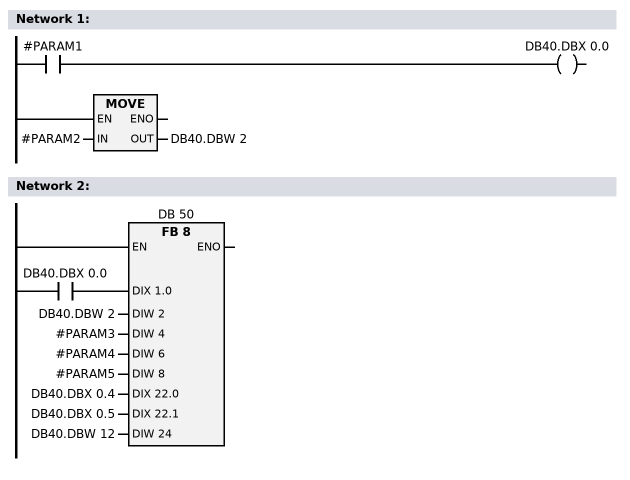
NETWORK
TITLE =
      A     #PARAM1;
      =     DB40.DBX 0.0;
      L     #PARAM2;
      T     DB40.DBW 2;
NETWORK
TITLE =
      A     DB40.DBX 0.0;
      =     L 0.0;
      BLD   103;
      CALL  FB 8 , DB 50 (
           DIX 1.0                  := L 0.0,
           DIW 2                    := DB40.DBW 2,
           DIW 4                    := #PARAM3,
           DIW 6                    := #PARAM4,
           DIW 8                    := #PARAM5,
           DIX 22.0                 := DB40.DBX 0.4,
           DIX 22.1                 := DB40.DBX 0.5,
           DIW 24                   := DB40.DBW 12);
      NOP   0;
NETWORK
TITLE =
      AN    DB40.DBX 0.4;
      JC    M001;
      L     DB40.DBW 16;
      +     1;
      T     DB40.DBW 16;
      NOP   0;
      NOP   0;
      NOP   0;
      BE;
M001: AN    DB40.DBX 0.5;
      BEC;
      L     DB40.DBW 18;
      +     1;
      T     DB40.DBW 18;
      L     DB40.DBW 12;
      T     DB40.DBW 14;
      NOP   0;
      NOP   0;
      NOP   0;
      BE;
NETWORK
TITLE =
END_FUNCTION

FUNCTION FC 31 : VOID
VERSION : 0.1
BEGIN
// (block stored without names or comments; labels and parameter names are numbered)
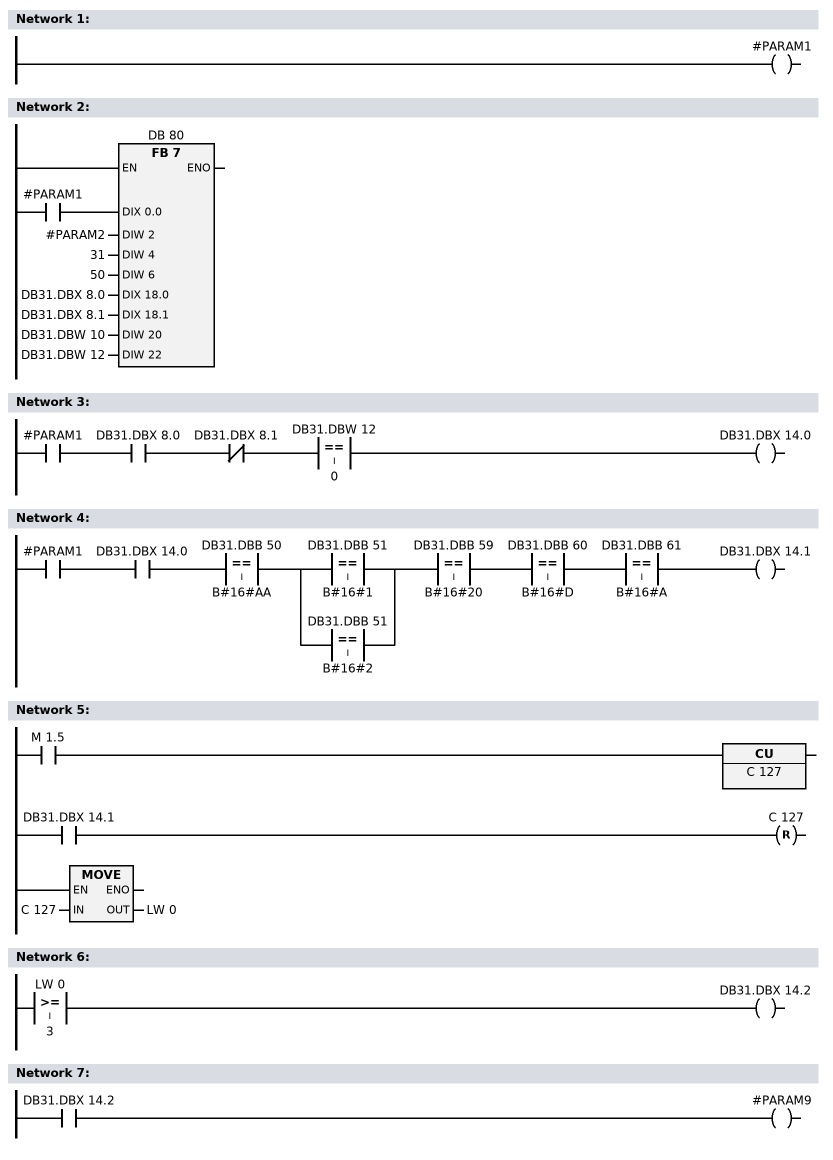
NETWORK
TITLE =
      SET;
      =     #PARAM1;
NETWORK
TITLE =
      A     #PARAM1;
      =     L 4.0;
      BLD   103;
      CALL  FB 7 , DB 80 (
           DIX 0.0                  := L 4.0,
           DIW 2                    := #PARAM2,
           DIW 4                    := 31,
           DIW 6                    := 50,
           DIX 18.0                 := DB31.DBX 8.0,
           DIX 18.1                 := DB31.DBX 8.1,
           DIW 20                   := DB31.DBW 10,
           DIW 22                   := DB31.DBW 12);
      NOP   0;
NETWORK
TITLE =
      A     #PARAM1;
      A     DB31.DBX 8.0;
      AN    DB31.DBX 8.1;
      A(;
      L     DB31.DBW 12;
      L     0;
      ==I;
      );
      =     DB31.DBX 14.0;
NETWORK
TITLE =
      A     #PARAM1;
      A     DB31.DBX 14.0;
      A(;
      L     DB31.DBB 50;
      L     B#16#AA;
      ==I;
      );
      A(;
      O(;
      L     DB31.DBB 51;
      L     B#16#1;
      ==I;
      );
      O(;
      L     DB31.DBB 51;
      L     B#16#2;
      ==I;
      );
      );
      A(;
      L     DB31.DBB 59;
      L     B#16#20;
      ==I;
      );
      A(;
      L     DB31.DBB 60;
      L     B#16#D;
      ==I;
      );
      A(;
      L     DB31.DBB 61;
      L     B#16#A;
      ==I;
      );
      =     DB31.DBX 14.1;
NETWORK
TITLE =
      A     M 1.5;
      CU    C 127;
      BLD   101;
      NOP   0;
      NOP   0;
      A     DB31.DBX 14.1;
      R     C 127;
      L     C 127;
      T     LW 0;
      NOP   0;
      NOP   0;
NETWORK
TITLE =
      L     LW 0;
      L     3;
      >=I;
      =     DB31.DBX 14.2;
NETWORK
TITLE =
      A     DB31.DBX 14.2;
      =     #PARAM9;
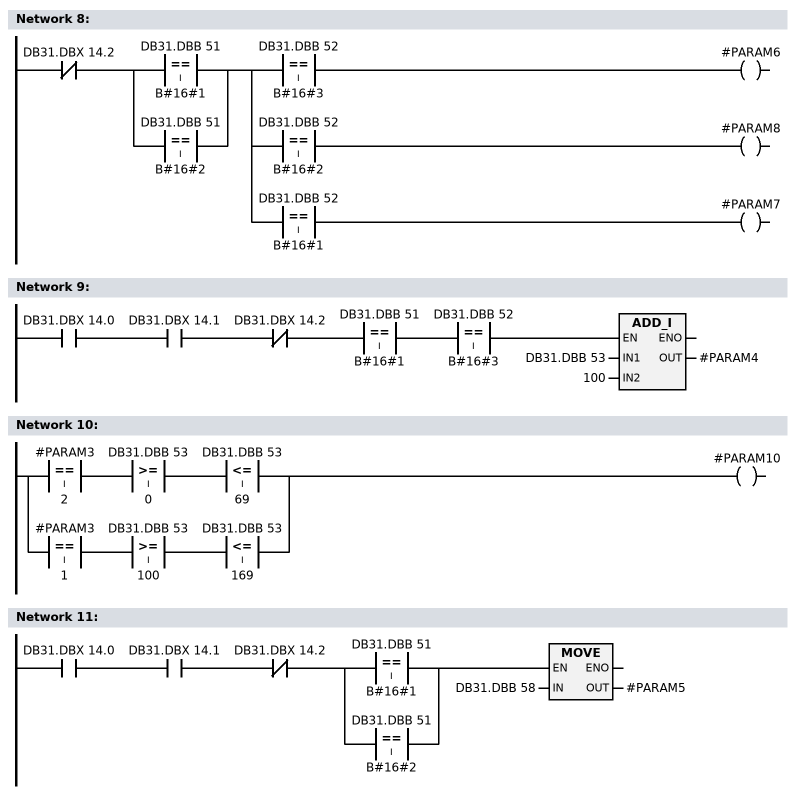
NETWORK
TITLE =
      AN    DB31.DBX 14.2;
      A(;
      O(;
      L     DB31.DBB 51;
      L     B#16#1;
      ==I;
      );
      O(;
      L     DB31.DBB 51;
      L     B#16#2;
      ==I;
      );
      );
      =     L 2.0;
      A     L 2.0;
      A(;
      L     DB31.DBB 52;
      L     B#16#3;
      ==I;
      );
      =     #PARAM6;
      A     L 2.0;
      A(;
      L     DB31.DBB 52;
      L     B#16#2;
      ==I;
      );
      =     #PARAM8;
      A     L 2.0;
      A(;
      L     DB31.DBB 52;
      L     B#16#1;
      ==I;
      );
      =     #PARAM7;
NETWORK
TITLE =
      A     DB31.DBX 14.0;
      A     DB31.DBX 14.1;
      AN    DB31.DBX 14.2;
      A(;
      L     DB31.DBB 51;
      L     B#16#1;
      ==I;
      );
      A(;
      L     DB31.DBB 52;
      L     B#16#3;
      ==I;
      );
      JNB   M001;
      L     DB31.DBB 53;
      L     100;
      +I;
      T     #PARAM4;
M001: NOP   0;
NETWORK
TITLE =
      A(;
      L     #PARAM3;
      L     2;
      ==I;
      );
      A(;
      L     DB31.DBB 53;
      L     0;
      >=I;
      );
      A(;
      L     DB31.DBB 53;
      L     69;
      <=I;
      );
      O;
      A(;
      L     #PARAM3;
      L     1;
      ==I;
      );
      A(;
      L     DB31.DBB 53;
      L     100;
      >=I;
      );
      A(;
      L     DB31.DBB 53;
      L     169;
      <=I;
      );
      =     #PARAM10;
NETWORK
TITLE =
      A     DB31.DBX 14.0;
      A     DB31.DBX 14.1;
      AN    DB31.DBX 14.2;
      A(;
      O(;
      L     DB31.DBB 51;
      L     B#16#1;
      ==I;
      );
      O(;
      L     DB31.DBB 51;
      L     B#16#2;
      ==I;
      );
      );
      JNB   M002;
      L     DB31.DBB 58;
      T     #PARAM5;
M002: NOP   0;
NETWORK
TITLE =
      A     DB31.DBX 8.0;
      JCN   M003;
      L     DB31.DBW 18;
      +     1;
      T     DB31.DBW 18;
      L     DB31.DBW 10;
      T     DB31.DBW 16;
      JU    M005;
M003: A     DB31.DBX 8.1;
      JCN   M004;
      L     DB31.DBW 20;
      +     1;
      T     DB31.DBW 20;
      L     0;
      L     DB31.DBW 12;
      ==I;
      JC    M005;
      T     DB31.DBW 22;
      JU    M005;
M004: L     0;
      L     DB31.DBW 12;
      ==I;
      JC    M005;
      T     DB31.DBW 22;
M005: CLR;
END_FUNCTION

FUNCTION FC 32 : VOID
VERSION : 0.1
BEGIN
// (block stored without names or comments; labels and parameter names are numbered)
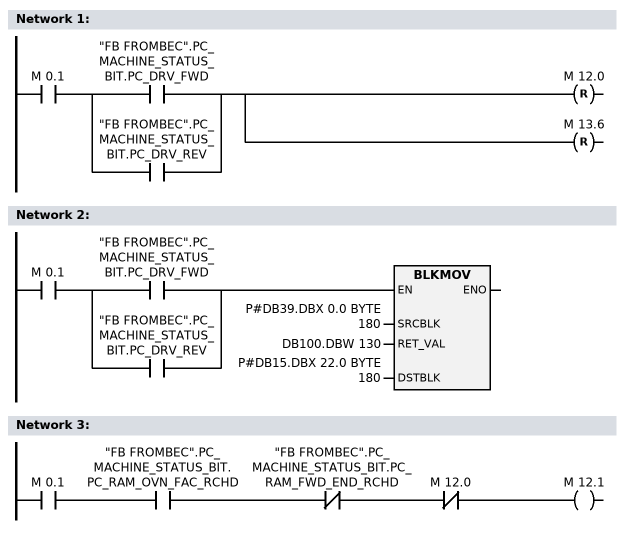
NETWORK
TITLE =
      A     M 0.1;
      A(;
      O     "FB FROMBEC".PC_MACHINE_STATUS_BIT.PC_DRV_FWD;
      O     "FB FROMBEC".PC_MACHINE_STATUS_BIT.PC_DRV_REV;
      );
      R     M 12.0;
      R     M 13.6;
NETWORK
TITLE =
      A     M 0.1;
      A(;
      O     "FB FROMBEC".PC_MACHINE_STATUS_BIT.PC_DRV_FWD;
      O     "FB FROMBEC".PC_MACHINE_STATUS_BIT.PC_DRV_REV;
      );
      JNB   M001;
      CALL  "BLKMOV" (
           SRCBLK                   := P#DB39.DBX 0.0 BYTE 180,
           RET_VAL                  := DB100.DBW 130,
           DSTBLK                   := P#DB15.DBX 22.0 BYTE 180);
M001: NOP   0;
NETWORK
TITLE =
      A     M 0.1;
      A     "FB FROMBEC".PC_MACHINE_STATUS_BIT.PC_RAM_OVN_FAC_RCHD;
      AN    "FB FROMBEC".PC_MACHINE_STATUS_BIT.PC_RAM_FWD_END_RCHD;
      AN    M 12.0;
      =     M 12.1;
NETWORK
TITLE =
      A(;
      A     M 0.1;
      A     M 12.1;
      A     M 1.3;
      FP    M 12.5;
      CU    C 120;
      BLD   101;
      NOP   0;
      NOP   0;
      A     M 12.0;
      R     C 120;
      L     C 120;
      T     MW 10;
      NOP   0;
      A     C 120;
      );
      A(;
      L     MW 10;
      L     91;
      ==I;
      );
      S     M 12.0;
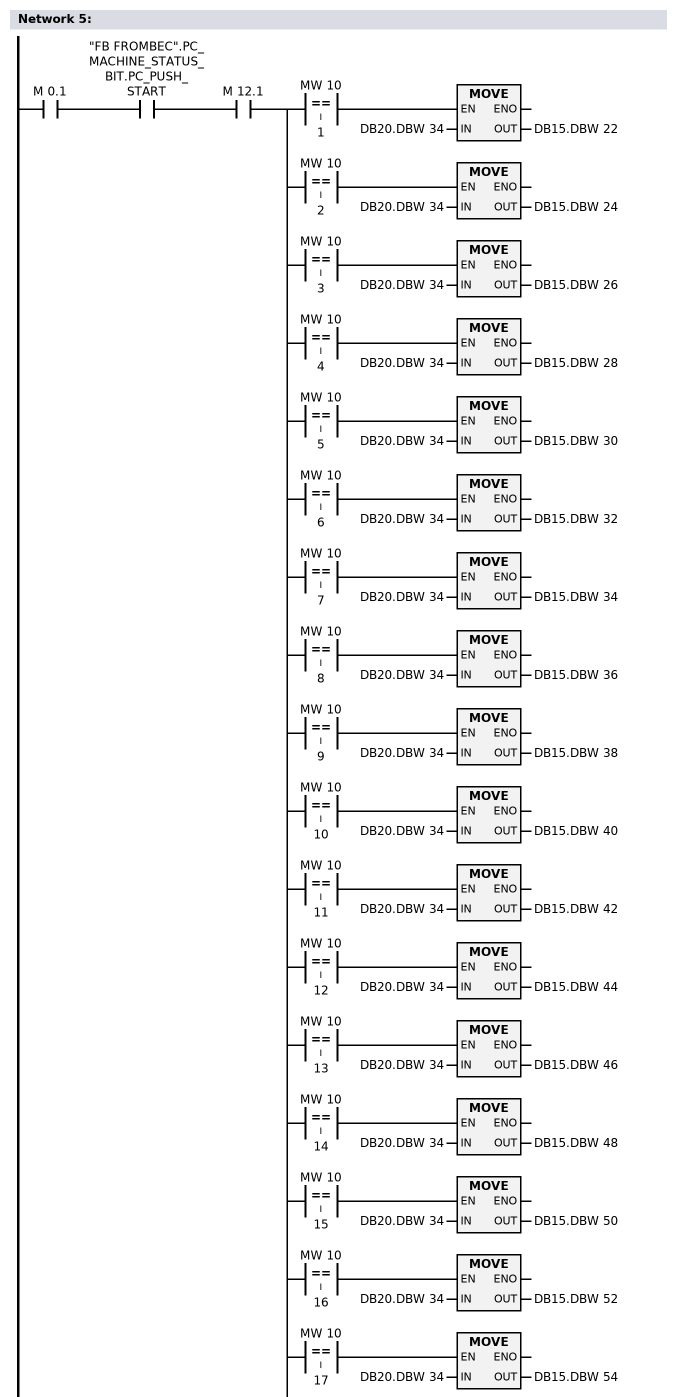
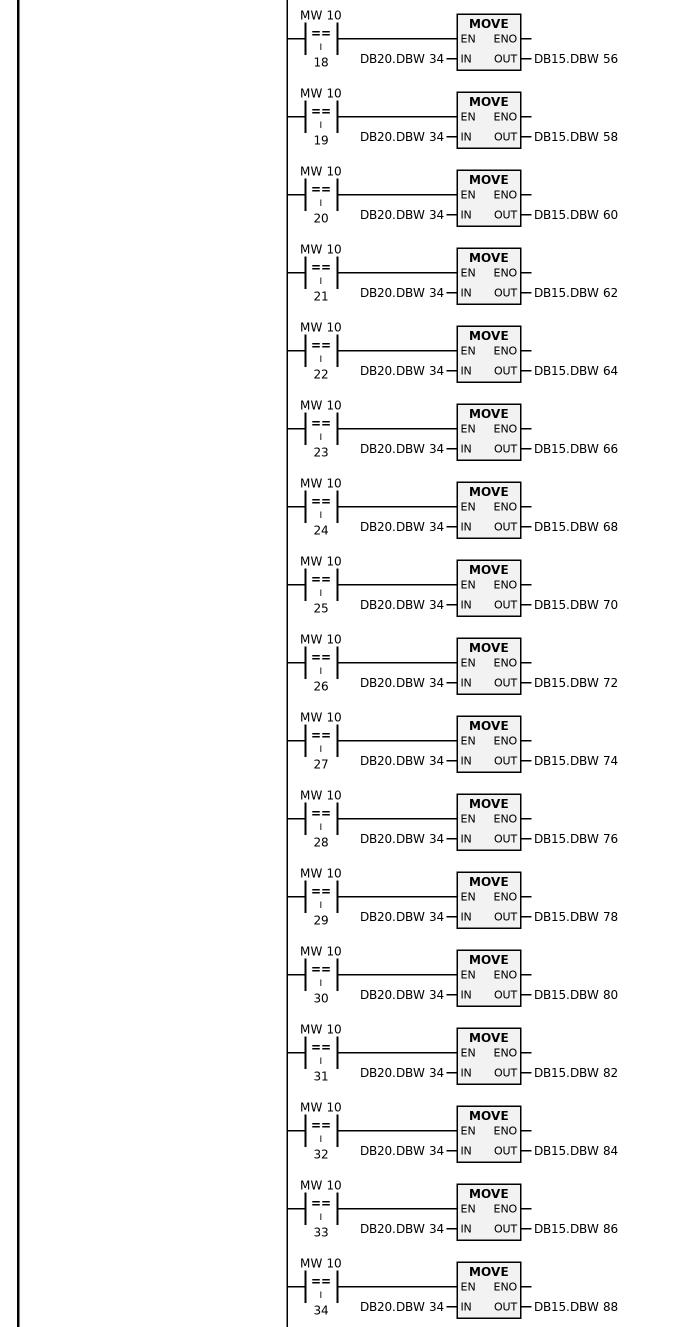
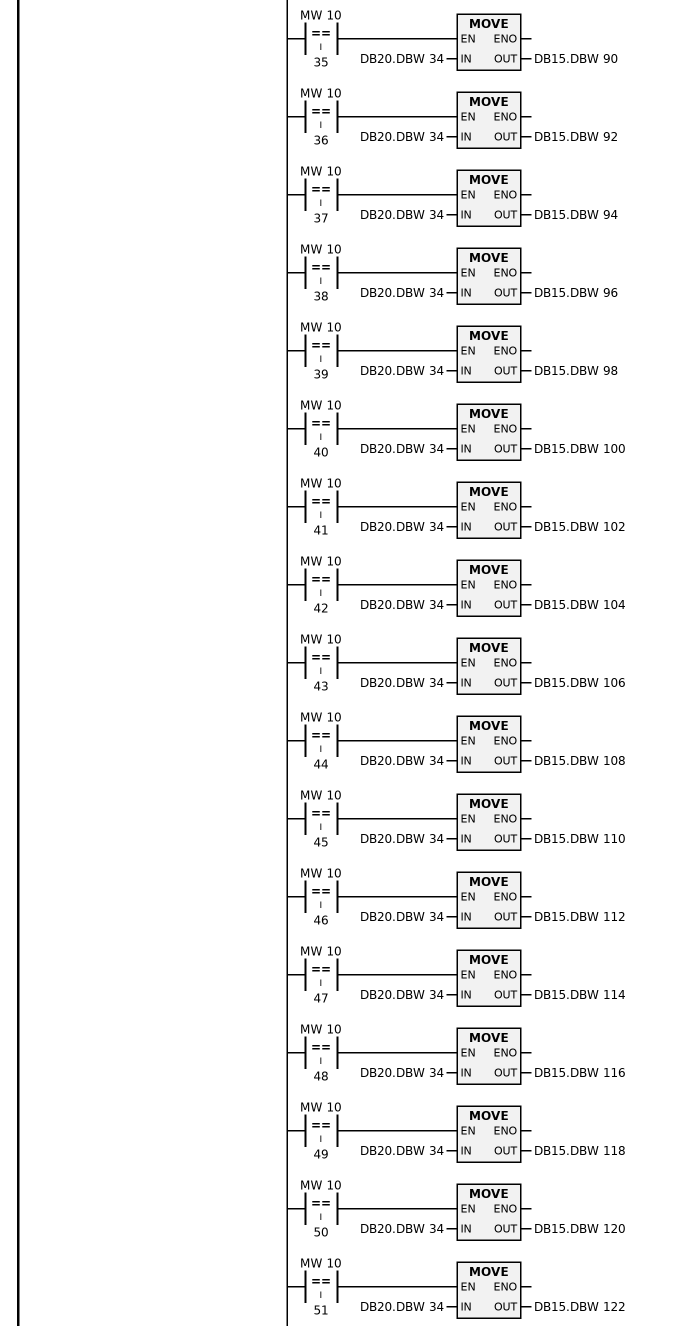
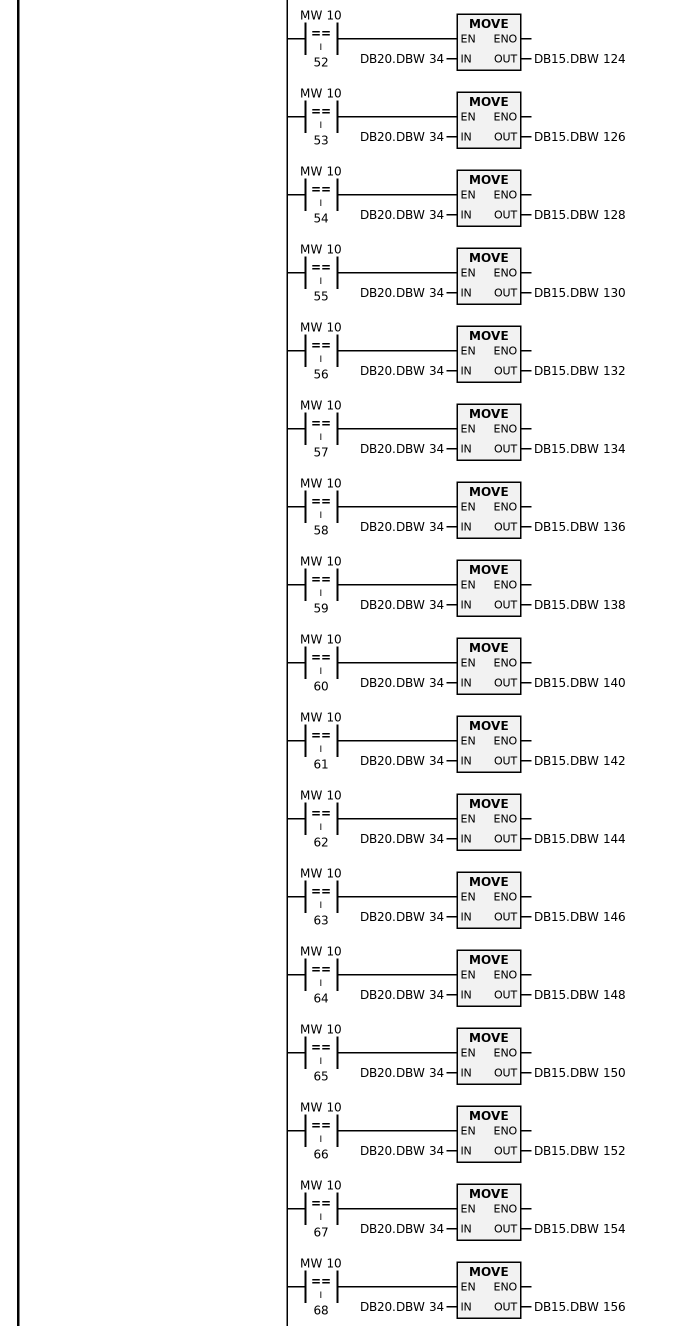
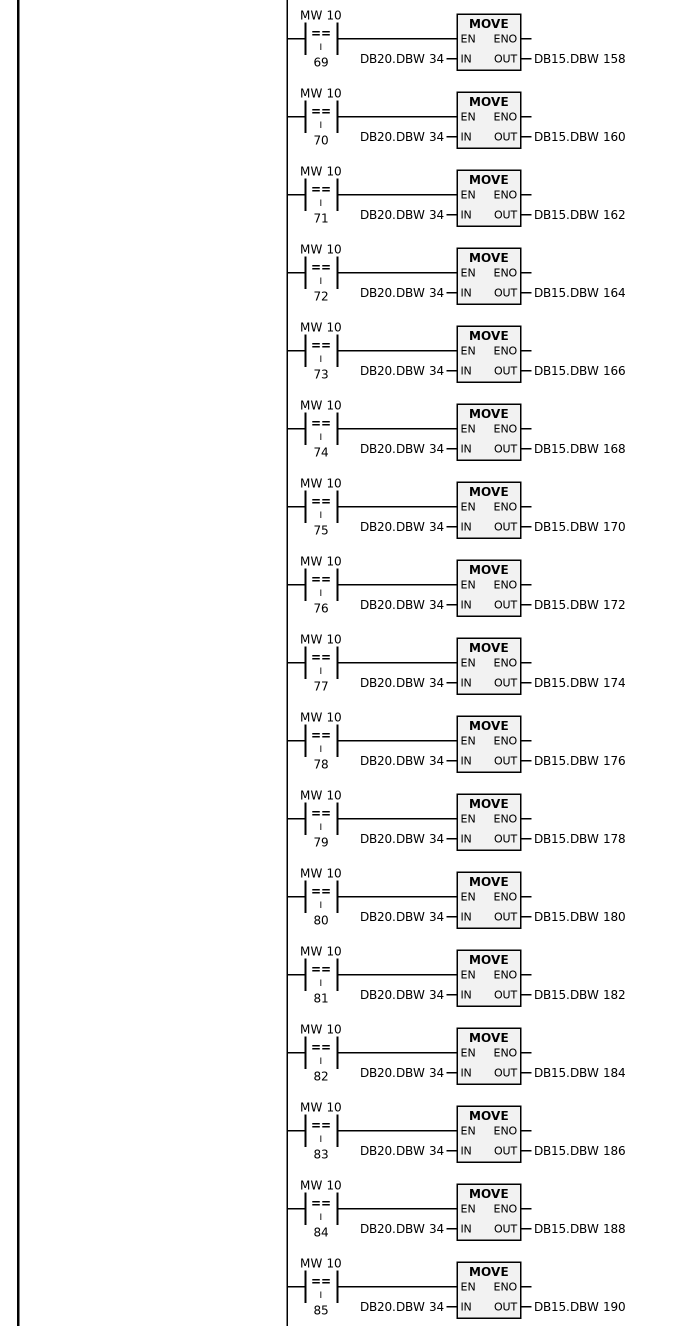
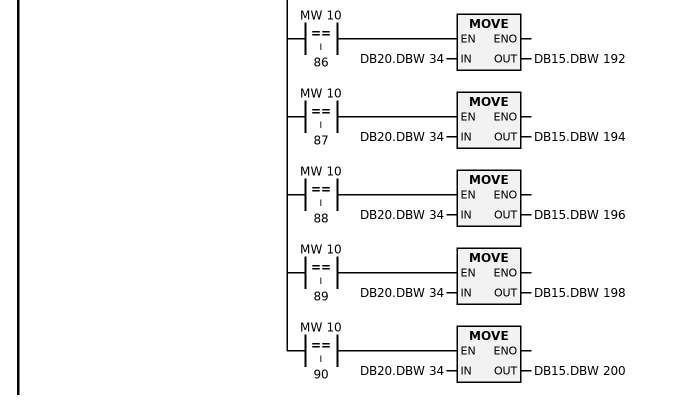
NETWORK
TITLE =
      A     M 0.1;
      A     "FB FROMBEC".PC_MACHINE_STATUS_BIT.PC_PUSH_START;
      A     M 12.1;
      =     L 12.0;
      A     L 12.0;
      A(;
      L     MW 10;
      L     1;
      ==I;
      );
      JNB   M002;
      L     DB20.DBW 34;
      T     DB15.DBW 22;
M002: NOP   0;
      A     L 12.0;
      A(;
      L     MW 10;
      L     2;
      ==I;
      );
      JNB   M003;
      L     DB20.DBW 34;
      T     DB15.DBW 24;
M003: NOP   0;
      A     L 12.0;
      A(;
      L     MW 10;
      L     3;
      ==I;
      );
      JNB   M004;
      L     DB20.DBW 34;
      T     DB15.DBW 26;
M004: NOP   0;
      A     L 12.0;
      A(;
      L     MW 10;
      L     4;
      ==I;
      );
      JNB   M005;
      L     DB20.DBW 34;
      T     DB15.DBW 28;
M005: NOP   0;
      A     L 12.0;
      A(;
      L     MW 10;
      L     5;
      ==I;
      );
      JNB   M006;
      L     DB20.DBW 34;
      T     DB15.DBW 30;
M006: NOP   0;
      A     L 12.0;
      A(;
      L     MW 10;
      L     6;
      ==I;
      );
      JNB   M007;
      L     DB20.DBW 34;
      T     DB15.DBW 32;
M007: NOP   0;
      A     L 12.0;
      A(;
      L     MW 10;
      L     7;
      ==I;
      );
      JNB   M008;
      L     DB20.DBW 34;
      T     DB15.DBW 34;
M008: NOP   0;
      A     L 12.0;
      A(;
      L     MW 10;
      L     8;
      ==I;
      );
      JNB   M009;
      L     DB20.DBW 34;
      T     DB15.DBW 36;
M009: NOP   0;
      A     L 12.0;
      A(;
      L     MW 10;
      L     9;
      ==I;
      );
      JNB   M010;
      L     DB20.DBW 34;
      T     DB15.DBW 38;
M010: NOP   0;
      A     L 12.0;
      A(;
      L     MW 10;
      L     10;
      ==I;
      );
      JNB   M011;
      L     DB20.DBW 34;
      T     DB15.DBW 40;
M011: NOP   0;
      A     L 12.0;
      A(;
      L     MW 10;
      L     11;
      ==I;
      );
      JNB   M012;
      L     DB20.DBW 34;
      T     DB15.DBW 42;
M012: NOP   0;
      A     L 12.0;
      A(;
      L     MW 10;
      L     12;
      ==I;
      );
      JNB   M013;
      L     DB20.DBW 34;
      T     DB15.DBW 44;
M013: NOP   0;
      A     L 12.0;
      A(;
      L     MW 10;
      L     13;
      ==I;
      );
      JNB   M014;
      L     DB20.DBW 34;
      T     DB15.DBW 46;
M014: NOP   0;
      A     L 12.0;
      A(;
      L     MW 10;
      L     14;
      ==I;
      );
      JNB   M015;
      L     DB20.DBW 34;
      T     DB15.DBW 48;
M015: NOP   0;
      A     L 12.0;
      A(;
      L     MW 10;
      L     15;
      ==I;
      );
      JNB   M016;
      L     DB20.DBW 34;
      T     DB15.DBW 50;
M016: NOP   0;
      A     L 12.0;
      A(;
      L     MW 10;
      L     16;
      ==I;
      );
      JNB   M017;
      L     DB20.DBW 34;
      T     DB15.DBW 52;
M017: NOP   0;
      A     L 12.0;
      A(;
      L     MW 10;
      L     17;
      ==I;
      );
      JNB   M018;
      L     DB20.DBW 34;
      T     DB15.DBW 54;
M018: NOP   0;
      A     L 12.0;
      A(;
      L     MW 10;
      L     18;
      ==I;
      );
      JNB   M019;
      L     DB20.DBW 34;
      T     DB15.DBW 56;
M019: NOP   0;
      A     L 12.0;
      A(;
      L     MW 10;
      L     19;
      ==I;
      );
      JNB   M020;
      L     DB20.DBW 34;
      T     DB15.DBW 58;
M020: NOP   0;
      A     L 12.0;
      A(;
      L     MW 10;
      L     20;
      ==I;
      );
      JNB   M021;
      L     DB20.DBW 34;
      T     DB15.DBW 60;
M021: NOP   0;
      A     L 12.0;
      A(;
      L     MW 10;
      L     21;
      ==I;
      );
      JNB   M022;
      L     DB20.DBW 34;
      T     DB15.DBW 62;
M022: NOP   0;
      A     L 12.0;
      A(;
      L     MW 10;
      L     22;
      ==I;
      );
      JNB   M023;
      L     DB20.DBW 34;
      T     DB15.DBW 64;
M023: NOP   0;
      A     L 12.0;
      A(;
      L     MW 10;
      L     23;
      ==I;
      );
      JNB   M024;
      L     DB20.DBW 34;
      T     DB15.DBW 66;
M024: NOP   0;
      A     L 12.0;
      A(;
      L     MW 10;
      L     24;
      ==I;
      );
      JNB   M025;
      L     DB20.DBW 34;
      T     DB15.DBW 68;
M025: NOP   0;
      A     L 12.0;
      A(;
      L     MW 10;
      L     25;
      ==I;
      );
      JNB   M026;
      L     DB20.DBW 34;
      T     DB15.DBW 70;
M026: NOP   0;
      A     L 12.0;
      A(;
      L     MW 10;
      L     26;
      ==I;
      );
      JNB   M027;
      L     DB20.DBW 34;
      T     DB15.DBW 72;
M027: NOP   0;
      A     L 12.0;
      A(;
      L     MW 10;
      L     27;
      ==I;
      );
      JNB   M028;
      L     DB20.DBW 34;
      T     DB15.DBW 74;
M028: NOP   0;
      A     L 12.0;
      A(;
      L     MW 10;
      L     28;
      ==I;
      );
      JNB   M029;
      L     DB20.DBW 34;
      T     DB15.DBW 76;
M029: NOP   0;
      A     L 12.0;
      A(;
      L     MW 10;
      L     29;
      ==I;
      );
      JNB   M030;
      L     DB20.DBW 34;
      T     DB15.DBW 78;
M030: NOP   0;
      A     L 12.0;
      A(;
      L     MW 10;
      L     30;
      ==I;
      );
      JNB   M031;
      L     DB20.DBW 34;
      T     DB15.DBW 80;
M031: NOP   0;
      A     L 12.0;
      A(;
      L     MW 10;
      L     31;
      ==I;
      );
      JNB   M032;
      L     DB20.DBW 34;
      T     DB15.DBW 82;
M032: NOP   0;
      A     L 12.0;
      A(;
      L     MW 10;
      L     32;
      ==I;
      );
      JNB   M033;
      L     DB20.DBW 34;
      T     DB15.DBW 84;
M033: NOP   0;
      A     L 12.0;
      A(;
      L     MW 10;
      L     33;
      ==I;
      );
      JNB   M034;
      L     DB20.DBW 34;
      T     DB15.DBW 86;
M034: NOP   0;
      A     L 12.0;
      A(;
      L     MW 10;
      L     34;
      ==I;
      );
      JNB   M035;
      L     DB20.DBW 34;
      T     DB15.DBW 88;
M035: NOP   0;
      A     L 12.0;
      A(;
      L     MW 10;
      L     35;
      ==I;
      );
      JNB   M036;
      L     DB20.DBW 34;
      T     DB15.DBW 90;
M036: NOP   0;
      A     L 12.0;
      A(;
      L     MW 10;
      L     36;
      ==I;
      );
      JNB   M037;
      L     DB20.DBW 34;
      T     DB15.DBW 92;
M037: NOP   0;
      A     L 12.0;
      A(;
      L     MW 10;
      L     37;
      ==I;
      );
      JNB   M038;
      L     DB20.DBW 34;
      T     DB15.DBW 94;
M038: NOP   0;
      A     L 12.0;
      A(;
      L     MW 10;
      L     38;
      ==I;
      );
      JNB   M039;
      L     DB20.DBW 34;
      T     DB15.DBW 96;
M039: NOP   0;
      A     L 12.0;
      A(;
      L     MW 10;
      L     39;
      ==I;
      );
      JNB   M040;
      L     DB20.DBW 34;
      T     DB15.DBW 98;
M040: NOP   0;
      A     L 12.0;
      A(;
      L     MW 10;
      L     40;
      ==I;
      );
      JNB   M041;
      L     DB20.DBW 34;
      T     DB15.DBW 100;
M041: NOP   0;
      A     L 12.0;
      A(;
      L     MW 10;
      L     41;
      ==I;
      );
      JNB   M042;
      L     DB20.DBW 34;
      T     DB15.DBW 102;
M042: NOP   0;
      A     L 12.0;
      A(;
      L     MW 10;
      L     42;
      ==I;
      );
      JNB   M043;
      L     DB20.DBW 34;
      T     DB15.DBW 104;
M043: NOP   0;
      A     L 12.0;
      A(;
      L     MW 10;
      L     43;
      ==I;
      );
      JNB   M044;
      L     DB20.DBW 34;
      T     DB15.DBW 106;
M044: NOP   0;
      A     L 12.0;
      A(;
      L     MW 10;
      L     44;
      ==I;
      );
      JNB   M045;
      L     DB20.DBW 34;
      T     DB15.DBW 108;
M045: NOP   0;
      A     L 12.0;
      A(;
      L     MW 10;
      L     45;
      ==I;
      );
      JNB   M046;
      L     DB20.DBW 34;
      T     DB15.DBW 110;
M046: NOP   0;
      A     L 12.0;
      A(;
      L     MW 10;
      L     46;
      ==I;
      );
      JNB   M047;
      L     DB20.DBW 34;
      T     DB15.DBW 112;
M047: NOP   0;
      A     L 12.0;
      A(;
      L     MW 10;
      L     47;
      ==I;
      );
      JNB   M048;
      L     DB20.DBW 34;
      T     DB15.DBW 114;
M048: NOP   0;
      A     L 12.0;
      A(;
      L     MW 10;
      L     48;
      ==I;
      );
      JNB   M049;
      L     DB20.DBW 34;
      T     DB15.DBW 116;
M049: NOP   0;
      A     L 12.0;
      A(;
      L     MW 10;
      L     49;
      ==I;
      );
      JNB   M050;
      L     DB20.DBW 34;
      T     DB15.DBW 118;
M050: NOP   0;
      A     L 12.0;
      A(;
      L     MW 10;
      L     50;
      ==I;
      );
      JNB   M051;
      L     DB20.DBW 34;
      T     DB15.DBW 120;
M051: NOP   0;
      A     L 12.0;
      A(;
      L     MW 10;
      L     51;
      ==I;
      );
      JNB   M052;
      L     DB20.DBW 34;
      T     DB15.DBW 122;
M052: NOP   0;
      A     L 12.0;
      A(;
      L     MW 10;
      L     52;
      ==I;
      );
      JNB   M053;
      L     DB20.DBW 34;
      T     DB15.DBW 124;
M053: NOP   0;
      A     L 12.0;
      A(;
      L     MW 10;
      L     53;
      ==I;
      );
      JNB   M054;
      L     DB20.DBW 34;
      T     DB15.DBW 126;
M054: NOP   0;
      A     L 12.0;
      A(;
      L     MW 10;
      L     54;
      ==I;
      );
      JNB   M055;
      L     DB20.DBW 34;
      T     DB15.DBW 128;
M055: NOP   0;
      A     L 12.0;
      A(;
      L     MW 10;
      L     55;
      ==I;
      );
      JNB   M056;
      L     DB20.DBW 34;
      T     DB15.DBW 130;
M056: NOP   0;
      A     L 12.0;
      A(;
      L     MW 10;
      L     56;
      ==I;
      );
      JNB   M057;
      L     DB20.DBW 34;
      T     DB15.DBW 132;
M057: NOP   0;
      A     L 12.0;
      A(;
      L     MW 10;
      L     57;
      ==I;
      );
      JNB   M058;
      L     DB20.DBW 34;
      T     DB15.DBW 134;
M058: NOP   0;
      A     L 12.0;
      A(;
      L     MW 10;
      L     58;
      ==I;
      );
      JNB   M059;
      L     DB20.DBW 34;
      T     DB15.DBW 136;
M059: NOP   0;
      A     L 12.0;
      A(;
      L     MW 10;
      L     59;
      ==I;
      );
      JNB   M060;
      L     DB20.DBW 34;
      T     DB15.DBW 138;
M060: NOP   0;
      A     L 12.0;
      A(;
      L     MW 10;
      L     60;
      ==I;
      );
      JNB   M061;
      L     DB20.DBW 34;
      T     DB15.DBW 140;
M061: NOP   0;
      A     L 12.0;
      A(;
      L     MW 10;
      L     61;
      ==I;
      );
      JNB   M062;
      L     DB20.DBW 34;
      T     DB15.DBW 142;
M062: NOP   0;
      A     L 12.0;
      A(;
      L     MW 10;
      L     62;
      ==I;
      );
      JNB   M063;
      L     DB20.DBW 34;
      T     DB15.DBW 144;
M063: NOP   0;
      A     L 12.0;
      A(;
      L     MW 10;
      L     63;
      ==I;
      );
      JNB   M064;
      L     DB20.DBW 34;
      T     DB15.DBW 146;
M064: NOP   0;
      A     L 12.0;
      A(;
      L     MW 10;
      L     64;
      ==I;
      );
      JNB   M065;
      L     DB20.DBW 34;
      T     DB15.DBW 148;
M065: NOP   0;
      A     L 12.0;
      A(;
      L     MW 10;
      L     65;
      ==I;
      );
      JNB   M066;
      L     DB20.DBW 34;
      T     DB15.DBW 150;
M066: NOP   0;
      A     L 12.0;
      A(;
      L     MW 10;
      L     66;
      ==I;
      );
      JNB   M067;
      L     DB20.DBW 34;
      T     DB15.DBW 152;
M067: NOP   0;
      A     L 12.0;
      A(;
      L     MW 10;
      L     67;
      ==I;
      );
      JNB   M068;
      L     DB20.DBW 34;
      T     DB15.DBW 154;
M068: NOP   0;
      A     L 12.0;
      A(;
      L     MW 10;
      L     68;
      ==I;
      );
      JNB   M069;
      L     DB20.DBW 34;
      T     DB15.DBW 156;
M069: NOP   0;
      A     L 12.0;
      A(;
      L     MW 10;
      L     69;
      ==I;
      );
      JNB   M070;
      L     DB20.DBW 34;
      T     DB15.DBW 158;
M070: NOP   0;
      A     L 12.0;
      A(;
      L     MW 10;
      L     70;
      ==I;
      );
      JNB   M071;
      L     DB20.DBW 34;
      T     DB15.DBW 160;
M071: NOP   0;
      A     L 12.0;
      A(;
      L     MW 10;
      L     71;
      ==I;
      );
      JNB   M072;
      L     DB20.DBW 34;
      T     DB15.DBW 162;
M072: NOP   0;
      A     L 12.0;
      A(;
      L     MW 10;
      L     72;
      ==I;
      );
      JNB   M073;
      L     DB20.DBW 34;
      T     DB15.DBW 164;
M073: NOP   0;
      A     L 12.0;
      A(;
      L     MW 10;
      L     73;
      ==I;
      );
      JNB   M074;
      L     DB20.DBW 34;
      T     DB15.DBW 166;
M074: NOP   0;
      A     L 12.0;
      A(;
      L     MW 10;
      L     74;
      ==I;
      );
      JNB   M075;
      L     DB20.DBW 34;
      T     DB15.DBW 168;
M075: NOP   0;
      A     L 12.0;
      A(;
      L     MW 10;
      L     75;
      ==I;
      );
      JNB   M076;
      L     DB20.DBW 34;
      T     DB15.DBW 170;
M076: NOP   0;
      A     L 12.0;
      A(;
      L     MW 10;
      L     76;
      ==I;
      );
      JNB   M077;
      L     DB20.DBW 34;
      T     DB15.DBW 172;
M077: NOP   0;
      A     L 12.0;
      A(;
      L     MW 10;
      L     77;
      ==I;
      );
      JNB   M078;
      L     DB20.DBW 34;
      T     DB15.DBW 174;
M078: NOP   0;
      A     L 12.0;
      A(;
      L     MW 10;
      L     78;
      ==I;
      );
      JNB   M079;
      L     DB20.DBW 34;
      T     DB15.DBW 176;
M079: NOP   0;
      A     L 12.0;
      A(;
      L     MW 10;
      L     79;
      ==I;
      );
      JNB   M080;
      L     DB20.DBW 34;
      T     DB15.DBW 178;
M080: NOP   0;
      A     L 12.0;
      A(;
      L     MW 10;
      L     80;
      ==I;
      );
      JNB   M081;
      L     DB20.DBW 34;
      T     DB15.DBW 180;
M081: NOP   0;
      A     L 12.0;
      A(;
      L     MW 10;
      L     81;
      ==I;
      );
      JNB   M082;
      L     DB20.DBW 34;
      T     DB15.DBW 182;
M082: NOP   0;
      A     L 12.0;
      A(;
      L     MW 10;
      L     82;
      ==I;
      );
      JNB   M083;
      L     DB20.DBW 34;
      T     DB15.DBW 184;
M083: NOP   0;
      A     L 12.0;
      A(;
      L     MW 10;
      L     83;
      ==I;
      );
      JNB   M084;
      L     DB20.DBW 34;
      T     DB15.DBW 186;
M084: NOP   0;
      A     L 12.0;
      A(;
      L     MW 10;
      L     84;
      ==I;
      );
      JNB   M085;
      L     DB20.DBW 34;
      T     DB15.DBW 188;
M085: NOP   0;
      A     L 12.0;
      A(;
      L     MW 10;
      L     85;
      ==I;
      );
      JNB   M086;
      L     DB20.DBW 34;
      T     DB15.DBW 190;
M086: NOP   0;
      A     L 12.0;
      A(;
      L     MW 10;
      L     86;
      ==I;
      );
      JNB   M087;
      L     DB20.DBW 34;
      T     DB15.DBW 192;
M087: NOP   0;
      A     L 12.0;
      A(;
      L     MW 10;
      L     87;
      ==I;
      );
      JNB   M088;
      L     DB20.DBW 34;
      T     DB15.DBW 194;
M088: NOP   0;
      A     L 12.0;
      A(;
      L     MW 10;
      L     88;
      ==I;
      );
      JNB   M089;
      L     DB20.DBW 34;
      T     DB15.DBW 196;
M089: NOP   0;
      A     L 12.0;
      A(;
      L     MW 10;
      L     89;
      ==I;
      );
      JNB   M090;
      L     DB20.DBW 34;
      T     DB15.DBW 198;
M090: NOP   0;
      A     L 12.0;
      A(;
      L     MW 10;
      L     90;
      ==I;
      );
      JNB   M091;
      L     DB20.DBW 34;
      T     DB15.DBW 200;
M091: NOP   0;
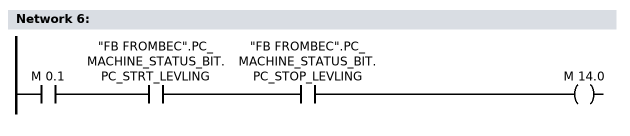
NETWORK
TITLE =
      A     M 0.1;
      A     "FB FROMBEC".PC_MACHINE_STATUS_BIT.PC_STRT_LEVLING;
      A     "FB FROMBEC".PC_MACHINE_STATUS_BIT.PC_STOP_LEVLING;
      =     M 14.0;
END_FUNCTION

FUNCTION FC 90 : VOID
AUTHOR : SKD
FAMILY : AuTiPosi
NAME : CDSPL
VERSION : 0.1
BEGIN
// (block stored without names or comments; labels and parameter names are numbered)
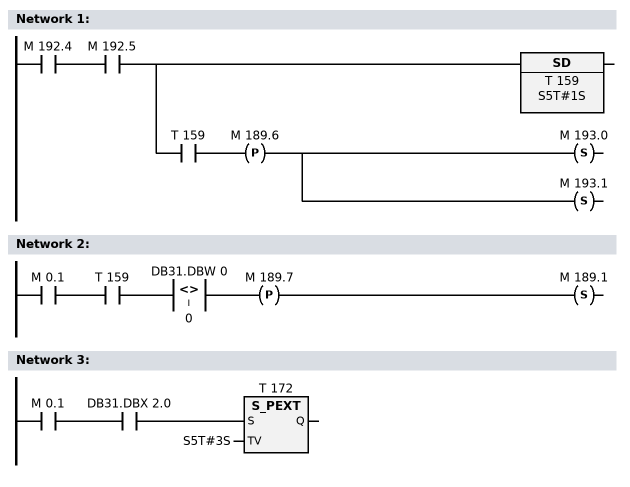
NETWORK
TITLE =
      A     M 192.4;
      A     M 192.5;
      =     L 0.0;
      A     L 0.0;
      BLD   102;
      L     S5T#1S;
      SD    T 159;
      A     L 0.0;
      A     T 159;
      FP    M 189.6;
      S     M 193.0;
      S     M 193.1;
NETWORK
TITLE =
      A     M 0.1;
      A     T 159;
      A(;
      L     DB31.DBW 0;
      L     0;
      <>I;
      );
      FP    M 189.7;
      S     M 189.1;
NETWORK
TITLE =
      A     M 0.1;
      A     DB31.DBX 2.0;
      L     S5T#3S;
      SE    T 172;
      NOP   0;
      NOP   0;
      NOP   0;
      NOP   0;
END_FUNCTION

FUNCTION FC 92 : VOID
AUTHOR : SKD
FAMILY : AuTiPosi
NAME : CDSPL
VERSION : 0.1
BEGIN
// (block stored without names or comments; labels and parameter names are numbered)
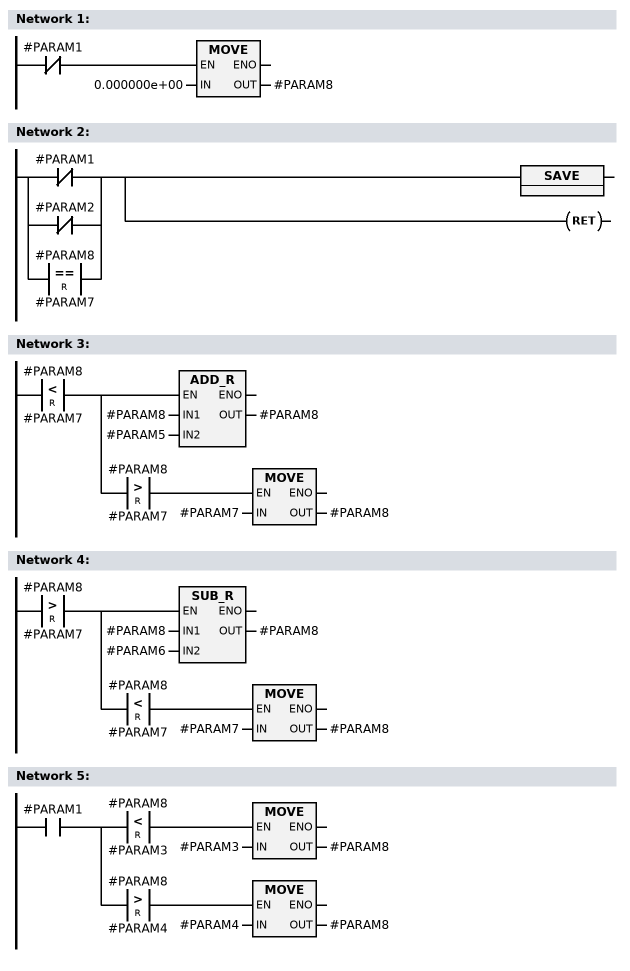
NETWORK
TITLE =
      AN    #PARAM1;
      JNB   M001;
      L     0.000000e+00;
      T     #PARAM8;
M001: NOP   0;
NETWORK
TITLE =
      ON    #PARAM1;
      ON    #PARAM2;
      O(;
      L     #PARAM8;
      L     #PARAM7;
      ==R;
      );
      SAVE;
      BEC;
NETWORK
TITLE =
      L     #PARAM8;
      L     #PARAM7;
      <R;
      =     L 0.0;
      A     L 0.0;
      JNB   M002;
      L     #PARAM8;
      L     #PARAM5;
      +R;
      T     #PARAM8;
M002: NOP   0;
      A     L 0.0;
      A(;
      L     #PARAM8;
      L     #PARAM7;
      >R;
      );
      JNB   M003;
      L     #PARAM7;
      T     #PARAM8;
M003: NOP   0;
NETWORK
TITLE =
      L     #PARAM8;
      L     #PARAM7;
      >R;
      =     L 0.0;
      A     L 0.0;
      JNB   M004;
      L     #PARAM8;
      L     #PARAM6;
      -R;
      T     #PARAM8;
M004: NOP   0;
      A     L 0.0;
      A(;
      L     #PARAM8;
      L     #PARAM7;
      <R;
      );
      JNB   M005;
      L     #PARAM7;
      T     #PARAM8;
M005: NOP   0;
NETWORK
TITLE =
      A     #PARAM1;
      =     L 0.0;
      A     L 0.0;
      A(;
      L     #PARAM8;
      L     #PARAM3;
      <R;
      );
      JNB   M006;
      L     #PARAM3;
      T     #PARAM8;
M006: NOP   0;
      A     L 0.0;
      A(;
      L     #PARAM8;
      L     #PARAM4;
      >R;
      );
      JNB   M007;
      L     #PARAM4;
      T     #PARAM8;
M007: NOP   0;
END_FUNCTION

FUNCTION FC 94 : VOID
AUTHOR : SKD
FAMILY : AuTiPosi
NAME : CDSPL
VERSION : 0.1
BEGIN
// (block stored without names or comments; labels and parameter names are numbered)
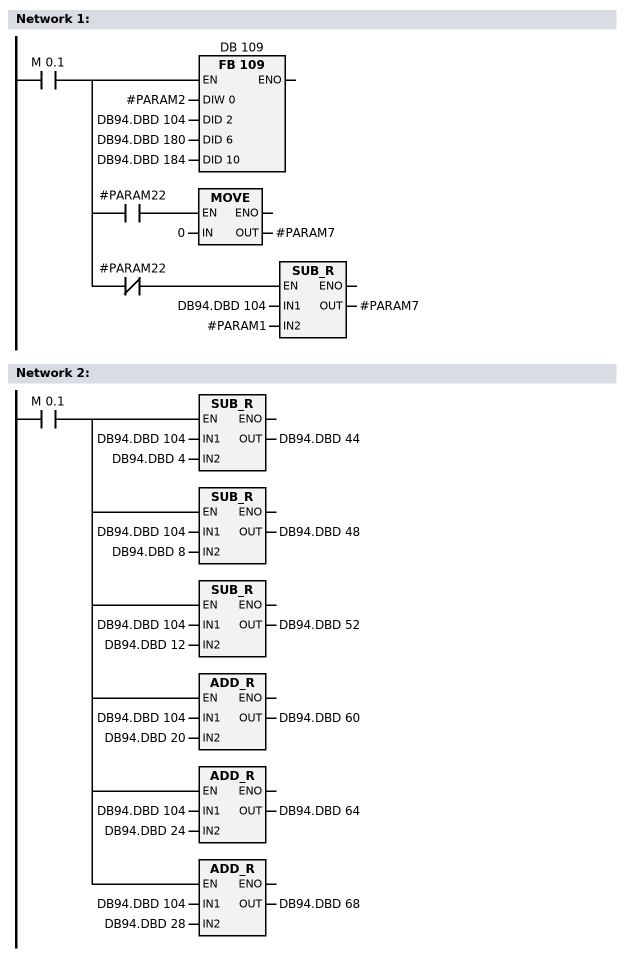
NETWORK
TITLE =
      A     M 0.1;
      =     L 6.0;
      A     L 6.0;
      JNB   M001;
      CALL  FB 109 , DB 109 (
           DIW 0                    := #PARAM2,
           DID 2                    := DB94.DBD 104,
           DID 6                    := DB94.DBD 180,
           DID 10                   := DB94.DBD 184);
M001: NOP   0;
      A     L 6.0;
      A     #PARAM22;
      JNB   M002;
      L     0;
      T     #PARAM7;
M002: NOP   0;
      A     L 6.0;
      AN    #PARAM22;
      JNB   M003;
      L     DB94.DBD 104;
      L     #PARAM1;
      -R;
      T     #PARAM7;
M003: NOP   0;
NETWORK
TITLE =
      A     M 0.1;
      =     L 6.0;
      A     L 6.0;
      JNB   M004;
      L     DB94.DBD 104;
      L     DB94.DBD 4;
      -R;
      T     DB94.DBD 44;
M004: NOP   0;
      A     L 6.0;
      JNB   M005;
      L     DB94.DBD 104;
      L     DB94.DBD 8;
      -R;
      T     DB94.DBD 48;
M005: NOP   0;
      A     L 6.0;
      JNB   M006;
      L     DB94.DBD 104;
      L     DB94.DBD 12;
      -R;
      T     DB94.DBD 52;
M006: NOP   0;
      A     L 6.0;
      JNB   M007;
      L     DB94.DBD 104;
      L     DB94.DBD 20;
      +R;
      T     DB94.DBD 60;
M007: NOP   0;
      A     L 6.0;
      JNB   M008;
      L     DB94.DBD 104;
      L     DB94.DBD 24;
      +R;
      T     DB94.DBD 64;
M008: NOP   0;
      A     L 6.0;
      JNB   M009;
      L     DB94.DBD 104;
      L     DB94.DBD 28;
      +R;
      T     DB94.DBD 68;
M009: NOP   0;
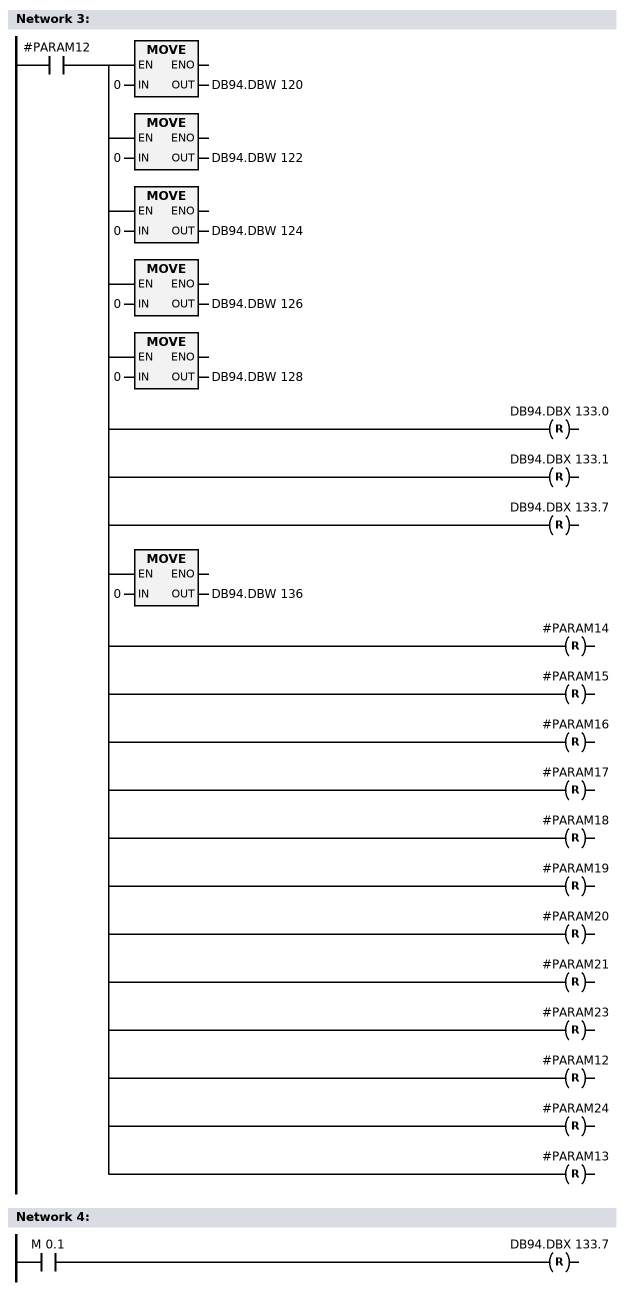
NETWORK
TITLE =
      A     #PARAM12;
      =     L 6.0;
      A     L 6.0;
      JNB   M010;
      L     0;
      T     DB94.DBW 120;
M010: NOP   0;
      A     L 6.0;
      JNB   M011;
      L     0;
      T     DB94.DBW 122;
M011: NOP   0;
      A     L 6.0;
      JNB   M012;
      L     0;
      T     DB94.DBW 124;
M012: NOP   0;
      A     L 6.0;
      JNB   M013;
      L     0;
      T     DB94.DBW 126;
M013: NOP   0;
      A     L 6.0;
      JNB   M014;
      L     0;
      T     DB94.DBW 128;
M014: NOP   0;
      A     L 6.0;
      BLD   102;
      R     DB94.DBX 133.0;
      A     L 6.0;
      BLD   102;
      R     DB94.DBX 133.1;
      A     L 6.0;
      BLD   102;
      R     DB94.DBX 133.7;
      A     L 6.0;
      JNB   M015;
      L     0;
      T     DB94.DBW 136;
M015: NOP   0;
      A     L 6.0;
      BLD   102;
      R     #PARAM14;
      A     L 6.0;
      BLD   102;
      R     #PARAM15;
      A     L 6.0;
      BLD   102;
      R     #PARAM16;
      A     L 6.0;
      BLD   102;
      R     #PARAM17;
      A     L 6.0;
      BLD   102;
      R     #PARAM18;
      A     L 6.0;
      BLD   102;
      R     #PARAM19;
      A     L 6.0;
      BLD   102;
      R     #PARAM20;
      A     L 6.0;
      BLD   102;
      R     #PARAM21;
      A     L 6.0;
      BLD   102;
      R     #PARAM23;
      A     L 6.0;
      BLD   102;
      R     #PARAM12;
      A     L 6.0;
      BLD   102;
      R     #PARAM24;
      A     L 6.0;
      BLD   102;
      R     #PARAM13;
NETWORK
TITLE =
      A     M 0.1;
      R     DB94.DBX 133.7;
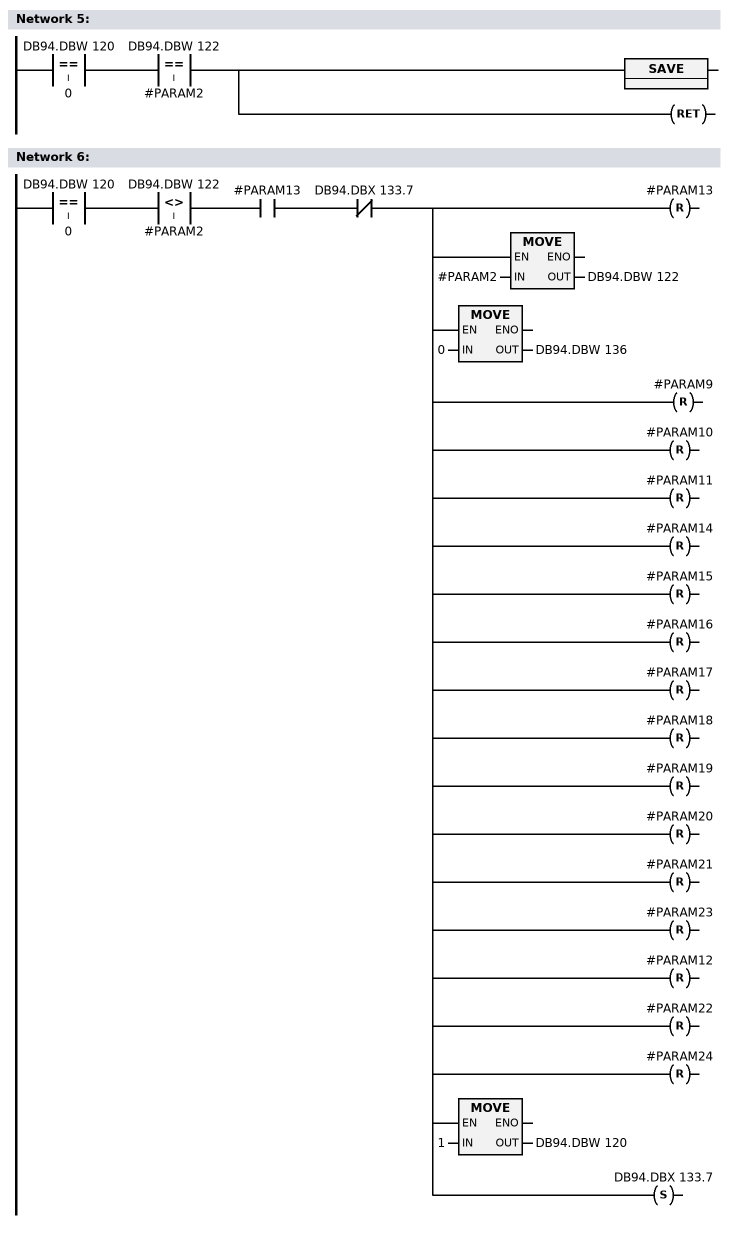
NETWORK
TITLE =
      A(;
      L     DB94.DBW 120;
      L     0;
      ==I;
      );
      A(;
      L     DB94.DBW 122;
      L     #PARAM2;
      ==I;
      );
      SAVE;
      BEC;
NETWORK
TITLE =
      A(;
      L     DB94.DBW 120;
      L     0;
      ==I;
      );
      A(;
      L     DB94.DBW 122;
      L     #PARAM2;
      <>I;
      );
      A     #PARAM13;
      AN    DB94.DBX 133.7;
      =     L 6.0;
      A     L 6.0;
      BLD   102;
      R     #PARAM13;
      A     L 6.0;
      JNB   M016;
      L     #PARAM2;
      T     DB94.DBW 122;
M016: NOP   0;
      A     L 6.0;
      JNB   M017;
      L     0;
      T     DB94.DBW 136;
M017: NOP   0;
      A     L 6.0;
      BLD   102;
      R     #PARAM9;
      A     L 6.0;
      BLD   102;
      R     #PARAM10;
      A     L 6.0;
      BLD   102;
      R     #PARAM11;
      A     L 6.0;
      BLD   102;
      R     #PARAM14;
      A     L 6.0;
      BLD   102;
      R     #PARAM15;
      A     L 6.0;
      BLD   102;
      R     #PARAM16;
      A     L 6.0;
      BLD   102;
      R     #PARAM17;
      A     L 6.0;
      BLD   102;
      R     #PARAM18;
      A     L 6.0;
      BLD   102;
      R     #PARAM19;
      A     L 6.0;
      BLD   102;
      R     #PARAM20;
      A     L 6.0;
      BLD   102;
      R     #PARAM21;
      A     L 6.0;
      BLD   102;
      R     #PARAM23;
      A     L 6.0;
      BLD   102;
      R     #PARAM12;
      A     L 6.0;
      BLD   102;
      R     #PARAM22;
      A     L 6.0;
      BLD   102;
      R     #PARAM24;
      A     L 6.0;
      JNB   M018;
      L     1;
      T     DB94.DBW 120;
M018: NOP   0;
      A     L 6.0;
      BLD   102;
      S     DB94.DBX 133.7;
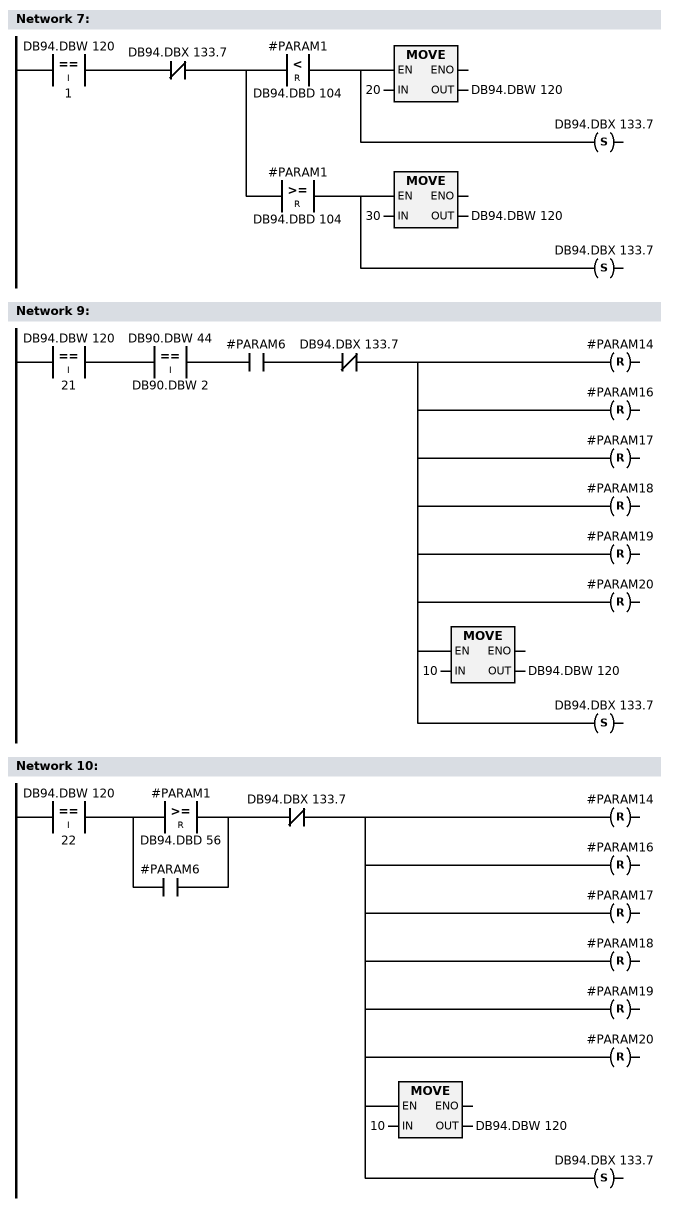
NETWORK
TITLE =
      A(;
      L     DB94.DBW 120;
      L     1;
      ==I;
      );
      AN    DB94.DBX 133.7;
      =     L 6.0;
      A     L 6.0;
      A(;
      L     #PARAM1;
      L     DB94.DBD 104;
      <R;
      );
      =     L 6.1;
      A     L 6.1;
      JNB   M019;
      L     20;
      T     DB94.DBW 120;
M019: NOP   0;
      A     L 6.1;
      BLD   102;
      S     DB94.DBX 133.7;
      A     L 6.0;
      A(;
      L     #PARAM1;
      L     DB94.DBD 104;
      >=R;
      );
      =     L 6.1;
      A     L 6.1;
      JNB   M020;
      L     30;
      T     DB94.DBW 120;
M020: NOP   0;
      A     L 6.1;
      BLD   102;
      S     DB94.DBX 133.7;
NETWORK
TITLE =
      A(;
      L     DB94.DBW 120;
      L     20;
      ==I;
      );
      AN    DB94.DBX 133.7;
      =     L 6.0;
      A     L 6.0;
      BLD   102;
      S     #PARAM14;
      A     L 6.0;
      BLD   102;
      R     #PARAM15;
      A     L 6.0;
      BLD   102;
      S     #PARAM16;
      A     L 6.0;
      BLD   102;
      R     #PARAM17;
      A     L 6.0;
      BLD   102;
      R     #PARAM18;
      A     L 6.0;
      BLD   102;
      R     #PARAM19;
      A     L 6.0;
      BLD   102;
      R     #PARAM20;
      A     L 6.0;
      A(;
      L     #PARAM1;
      L     DB94.DBD 44;
      >=R;
      );
      S     #PARAM17;
      R     #PARAM16;
      R     #PARAM18;
      R     #PARAM19;
      R     #PARAM20;
      A     L 6.0;
      A(;
      L     #PARAM1;
      L     DB94.DBD 48;
      >=R;
      );
      S     #PARAM18;
      R     #PARAM16;
      R     #PARAM17;
      R     #PARAM19;
      R     #PARAM20;
      A     L 6.0;
      A(;
      L     #PARAM1;
      L     DB94.DBD 52;
      >=R;
      );
      S     #PARAM19;
      R     #PARAM16;
      R     #PARAM17;
      R     #PARAM18;
      R     #PARAM20;
      A     L 6.0;
      A     #PARAM5;
      A(;
      O(;
      L     DB90.DBW 48;
      L     DB94.DBW 102;
      ==I;
      );
      O(;
      L     DB90.DBW 44;
      L     DB94.DBW 102;
      ==I;
      );
      );
      =     L 0.0;
      A     L 6.0;
      A     L 0.0;
      S     #PARAM21;
      S     #PARAM20;
      R     #PARAM16;
      R     #PARAM17;
      R     #PARAM18;
      R     #PARAM19;
      A     L 6.0;
      A     L 0.0;
      A(;
      L     DB94.DBD 16;
      L     0.000000e+00;
      ==R;
      );
      AN    DB94.DBX 133.7;
      =     L 6.1;
      A     L 6.1;
      JNB   M021;
      L     21;
      T     DB94.DBW 120;
M021: NOP   0;
      A     L 6.1;
      BLD   102;
      S     DB94.DBX 133.7;
      A     L 6.0;
      A     L 0.0;
      A(;
      L     DB94.DBD 16;
      L     0.000000e+00;
      <R;
      );
      AN    DB94.DBX 133.7;
      =     L 6.1;
      A     L 6.1;
      JNB   M022;
      L     22;
      T     DB94.DBW 120;
M022: NOP   0;
      A     L 6.1;
      BLD   102;
      S     DB94.DBX 133.7;
      A     L 6.0;
      A     L 0.0;
      A(;
      L     DB94.DBD 16;
      L     0.000000e+00;
      >R;
      );
      AN    DB94.DBX 133.7;
      =     L 6.1;
      A     L 6.1;
      JNB   M023;
      L     23;
      T     DB94.DBW 120;
M023: NOP   0;
      A     L 6.1;
      BLD   102;
      S     DB94.DBX 133.7;
      A     L 6.0;
      A     L 0.0;
      A(;
      O(;
      L     DB94.DBW 120;
      L     21;
      ==I;
      );
      O(;
      L     DB94.DBW 120;
      L     22;
      ==I;
      );
      O(;
      L     DB94.DBW 120;
      L     23;
      ==I;
      );
      );
      =     L 6.1;
      A     L 6.1;
      JNB   M024;
      L     #PARAM1;
      L     DB94.DBD 92;
      +R;
      T     LD 2;
M024: NOP   0;
      A     L 6.1;
      JNB   M025;
      L     LD 2;
      L     DB94.DBD 16;
      +R;
      T     DB94.DBD 56;
M025: NOP   0;
NETWORK
TITLE =
      A(;
      L     DB94.DBW 120;
      L     21;
      ==I;
      );
      A(;
      L     DB90.DBW 44;
      L     DB90.DBW 2;
      ==I;
      );
      A     #PARAM6;
      AN    DB94.DBX 133.7;
      =     L 6.0;
      A     L 6.0;
      BLD   102;
      R     #PARAM14;
      A     L 6.0;
      BLD   102;
      R     #PARAM16;
      A     L 6.0;
      BLD   102;
      R     #PARAM17;
      A     L 6.0;
      BLD   102;
      R     #PARAM18;
      A     L 6.0;
      BLD   102;
      R     #PARAM19;
      A     L 6.0;
      BLD   102;
      R     #PARAM20;
      A     L 6.0;
      JNB   M026;
      L     10;
      T     DB94.DBW 120;
M026: NOP   0;
      A     L 6.0;
      BLD   102;
      S     DB94.DBX 133.7;
NETWORK
TITLE =
      A(;
      L     DB94.DBW 120;
      L     22;
      ==I;
      );
      A(;
      O(;
      L     #PARAM1;
      L     DB94.DBD 56;
      >=R;
      );
      O     #PARAM6;
      );
      AN    DB94.DBX 133.7;
      =     L 6.0;
      A     L 6.0;
      BLD   102;
      R     #PARAM14;
      A     L 6.0;
      BLD   102;
      R     #PARAM16;
      A     L 6.0;
      BLD   102;
      R     #PARAM17;
      A     L 6.0;
      BLD   102;
      R     #PARAM18;
      A     L 6.0;
      BLD   102;
      R     #PARAM19;
      A     L 6.0;
      BLD   102;
      R     #PARAM20;
      A     L 6.0;
      JNB   M027;
      L     10;
      T     DB94.DBW 120;
M027: NOP   0;
      A     L 6.0;
      BLD   102;
      S     DB94.DBX 133.7;
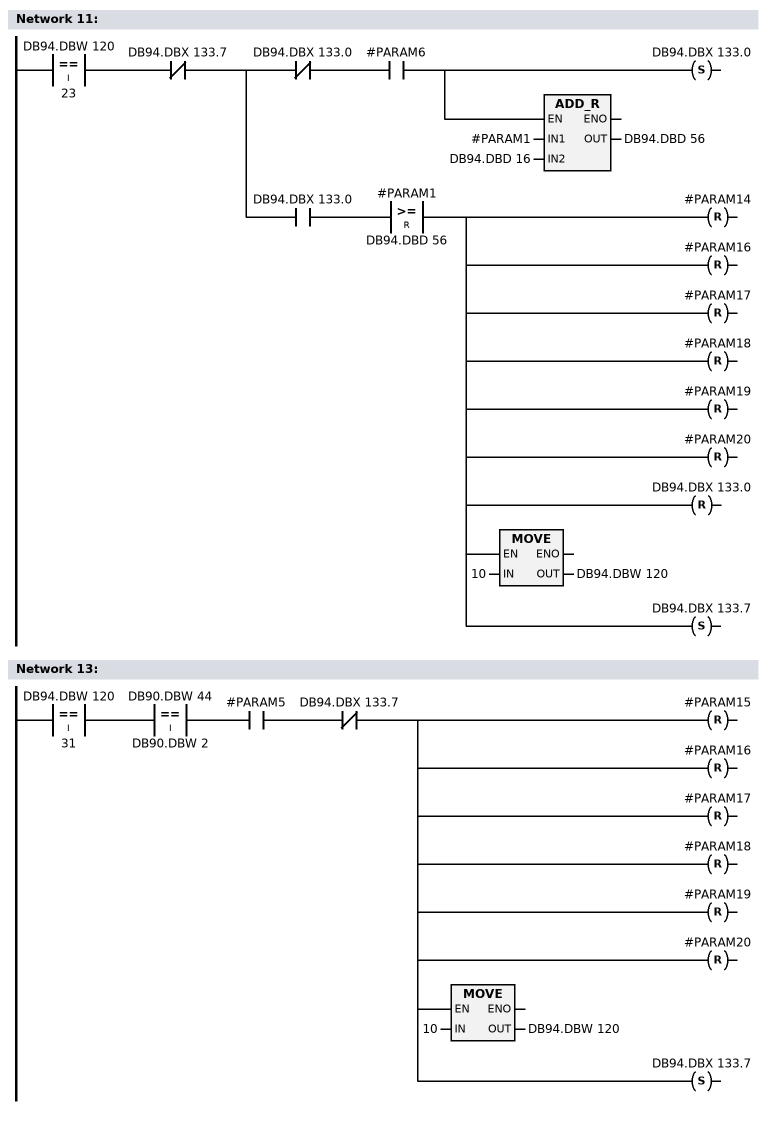
NETWORK
TITLE =
      A(;
      L     DB94.DBW 120;
      L     23;
      ==I;
      );
      AN    DB94.DBX 133.7;
      =     L 6.0;
      A     L 6.0;
      AN    DB94.DBX 133.0;
      A     #PARAM6;
      =     L 6.1;
      A     L 6.1;
      BLD   102;
      S     DB94.DBX 133.0;
      A     L 6.1;
      JNB   M028;
      L     #PARAM1;
      L     DB94.DBD 16;
      +R;
      T     DB94.DBD 56;
M028: NOP   0;
      A     L 6.0;
      A     DB94.DBX 133.0;
      A(;
      L     #PARAM1;
      L     DB94.DBD 56;
      >=R;
      );
      =     L 6.1;
      A     L 6.1;
      BLD   102;
      R     #PARAM14;
      A     L 6.1;
      BLD   102;
      R     #PARAM16;
      A     L 6.1;
      BLD   102;
      R     #PARAM17;
      A     L 6.1;
      BLD   102;
      R     #PARAM18;
      A     L 6.1;
      BLD   102;
      R     #PARAM19;
      A     L 6.1;
      BLD   102;
      R     #PARAM20;
      A     L 6.1;
      BLD   102;
      R     DB94.DBX 133.0;
      A     L 6.1;
      JNB   M029;
      L     10;
      T     DB94.DBW 120;
M029: NOP   0;
      A     L 6.1;
      BLD   102;
      S     DB94.DBX 133.7;
NETWORK
TITLE =
      A(;
      L     DB94.DBW 120;
      L     30;
      ==I;
      );
      AN    DB94.DBX 133.7;
      =     L 6.0;
      A     L 6.0;
      BLD   102;
      S     #PARAM15;
      A     L 6.0;
      BLD   102;
      R     #PARAM14;
      A     L 6.0;
      BLD   102;
      S     #PARAM16;
      A     L 6.0;
      BLD   102;
      R     #PARAM17;
      A     L 6.0;
      BLD   102;
      R     #PARAM18;
      A     L 6.0;
      BLD   102;
      R     #PARAM19;
      A     L 6.0;
      BLD   102;
      R     #PARAM20;
      A     L 6.0;
      A(;
      L     #PARAM1;
      L     DB94.DBD 60;
      <=R;
      );
      S     #PARAM17;
      R     #PARAM16;
      R     #PARAM18;
      R     #PARAM19;
      R     #PARAM20;
      A     L 6.0;
      A(;
      L     #PARAM1;
      L     DB94.DBD 64;
      <=R;
      );
      S     #PARAM18;
      R     #PARAM16;
      R     #PARAM17;
      R     #PARAM19;
      R     #PARAM20;
      A     L 6.0;
      A(;
      L     #PARAM1;
      L     DB94.DBD 68;
      <=R;
      );
      S     #PARAM19;
      R     #PARAM16;
      R     #PARAM17;
      R     #PARAM18;
      R     #PARAM20;
      A     L 6.0;
      A     #PARAM6;
      A(;
      O(;
      L     DB90.DBW 46;
      L     DB94.DBW 102;
      ==I;
      );
      O(;
      L     DB90.DBW 44;
      L     DB94.DBW 102;
      ==I;
      );
      );
      =     L 0.0;
      A     L 6.0;
      A     L 0.0;
      S     #PARAM21;
      S     #PARAM20;
      R     #PARAM16;
      R     #PARAM17;
      R     #PARAM18;
      R     #PARAM19;
      A     L 6.0;
      A     L 0.0;
      A(;
      L     DB94.DBD 32;
      L     0.000000e+00;
      ==R;
      );
      AN    DB94.DBX 133.7;
      =     L 6.1;
      A     L 6.1;
      JNB   M030;
      L     31;
      T     DB94.DBW 120;
M030: NOP   0;
      A     L 6.1;
      BLD   102;
      S     DB94.DBX 133.7;
      A     L 6.0;
      A     L 0.0;
      A(;
      L     DB94.DBD 32;
      L     0.000000e+00;
      <R;
      );
      AN    DB94.DBX 133.7;
      =     L 6.1;
      A     L 6.1;
      JNB   M031;
      L     32;
      T     DB94.DBW 120;
M031: NOP   0;
      A     L 6.1;
      BLD   102;
      S     DB94.DBX 133.7;
      A     L 6.0;
      A     L 0.0;
      A(;
      L     DB94.DBD 32;
      L     0.000000e+00;
      >R;
      );
      AN    DB94.DBX 133.7;
      =     L 6.1;
      A     L 6.1;
      JNB   M032;
      L     33;
      T     DB94.DBW 120;
M032: NOP   0;
      A     L 6.1;
      BLD   102;
      S     DB94.DBX 133.7;
      A     L 6.0;
      A     L 0.0;
      A(;
      O(;
      L     DB94.DBW 120;
      L     31;
      ==I;
      );
      O(;
      L     DB94.DBW 120;
      L     32;
      ==I;
      );
      O(;
      L     DB94.DBW 120;
      L     33;
      ==I;
      );
      );
      =     L 6.1;
      A     L 6.1;
      JNB   M033;
      L     #PARAM1;
      L     DB94.DBD 96;
      -R;
      T     LD 2;
M033: NOP   0;
      A     L 6.1;
      JNB   M034;
      L     LD 2;
      L     DB94.DBD 32;
      -R;
      T     DB94.DBD 72;
M034: NOP   0;
NETWORK
TITLE =
      A(;
      L     DB94.DBW 120;
      L     31;
      ==I;
      );
      A(;
      L     DB90.DBW 44;
      L     DB90.DBW 2;
      ==I;
      );
      A     #PARAM5;
      AN    DB94.DBX 133.7;
      =     L 6.0;
      A     L 6.0;
      BLD   102;
      R     #PARAM15;
      A     L 6.0;
      BLD   102;
      R     #PARAM16;
      A     L 6.0;
      BLD   102;
      R     #PARAM17;
      A     L 6.0;
      BLD   102;
      R     #PARAM18;
      A     L 6.0;
      BLD   102;
      R     #PARAM19;
      A     L 6.0;
      BLD   102;
      R     #PARAM20;
      A     L 6.0;
      JNB   M035;
      L     10;
      T     DB94.DBW 120;
M035: NOP   0;
      A     L 6.0;
      BLD   102;
      S     DB94.DBX 133.7;
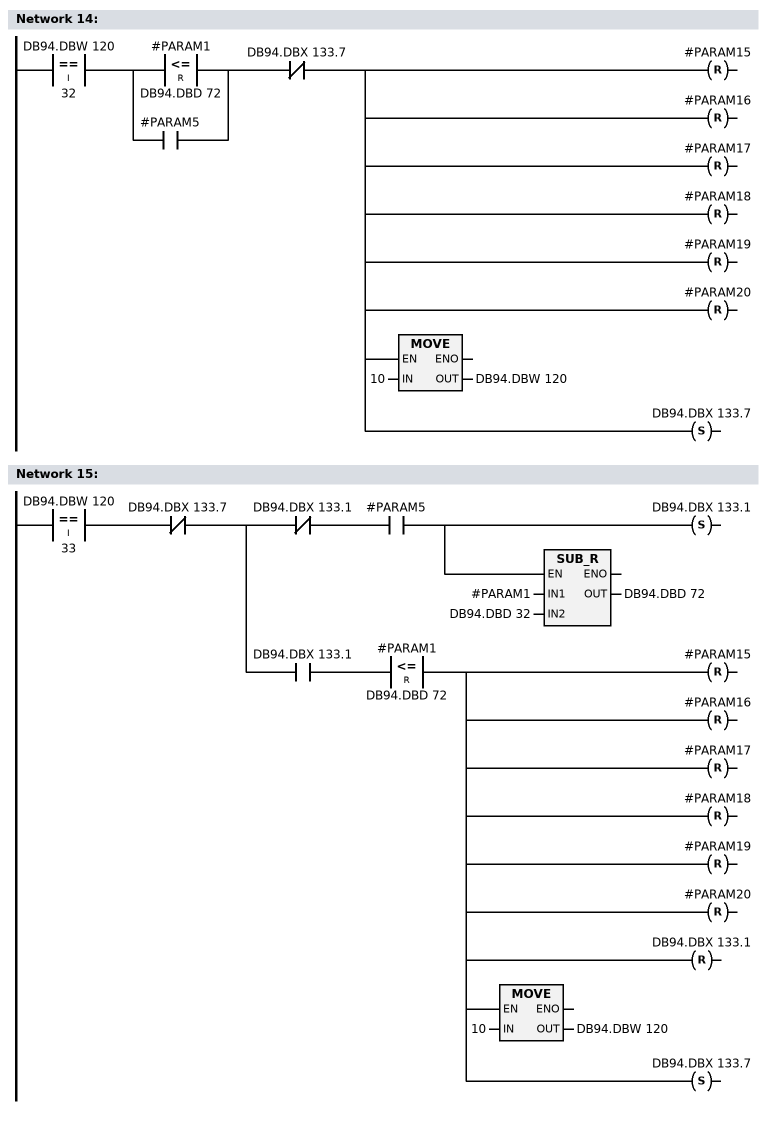
NETWORK
TITLE =
      A(;
      L     DB94.DBW 120;
      L     32;
      ==I;
      );
      A(;
      O(;
      L     #PARAM1;
      L     DB94.DBD 72;
      <=R;
      );
      O     #PARAM5;
      );
      AN    DB94.DBX 133.7;
      =     L 6.0;
      A     L 6.0;
      BLD   102;
      R     #PARAM15;
      A     L 6.0;
      BLD   102;
      R     #PARAM16;
      A     L 6.0;
      BLD   102;
      R     #PARAM17;
      A     L 6.0;
      BLD   102;
      R     #PARAM18;
      A     L 6.0;
      BLD   102;
      R     #PARAM19;
      A     L 6.0;
      BLD   102;
      R     #PARAM20;
      A     L 6.0;
      JNB   M036;
      L     10;
      T     DB94.DBW 120;
M036: NOP   0;
      A     L 6.0;
      BLD   102;
      S     DB94.DBX 133.7;
NETWORK
TITLE =
      A(;
      L     DB94.DBW 120;
      L     33;
      ==I;
      );
      AN    DB94.DBX 133.7;
      =     L 6.0;
      A     L 6.0;
      AN    DB94.DBX 133.1;
      A     #PARAM5;
      =     L 6.1;
      A     L 6.1;
      BLD   102;
      S     DB94.DBX 133.1;
      A     L 6.1;
      JNB   M037;
      L     #PARAM1;
      L     DB94.DBD 32;
      -R;
      T     DB94.DBD 72;
M037: NOP   0;
      A     L 6.0;
      A     DB94.DBX 133.1;
      A(;
      L     #PARAM1;
      L     DB94.DBD 72;
      <=R;
      );
      =     L 6.1;
      A     L 6.1;
      BLD   102;
      R     #PARAM15;
      A     L 6.1;
      BLD   102;
      R     #PARAM16;
      A     L 6.1;
      BLD   102;
      R     #PARAM17;
      A     L 6.1;
      BLD   102;
      R     #PARAM18;
      A     L 6.1;
      BLD   102;
      R     #PARAM19;
      A     L 6.1;
      BLD   102;
      R     #PARAM20;
      A     L 6.1;
      BLD   102;
      R     DB94.DBX 133.1;
      A     L 6.1;
      JNB   M038;
      L     10;
      T     DB94.DBW 120;
M038: NOP   0;
      A     L 6.1;
      BLD   102;
      S     DB94.DBX 133.7;
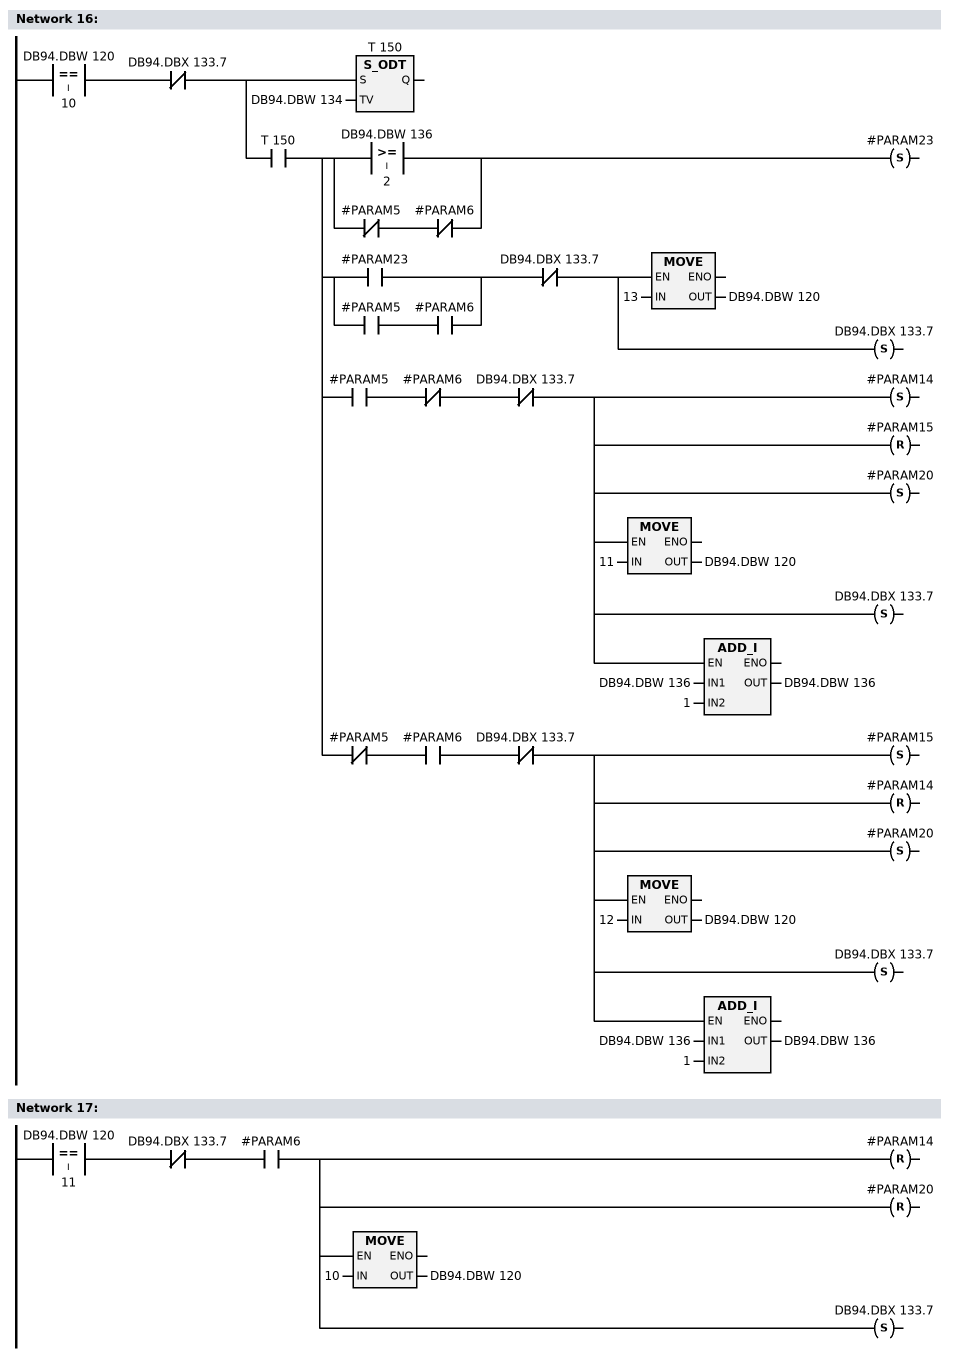
NETWORK
TITLE =
      A(;
      L     DB94.DBW 120;
      L     10;
      ==I;
      );
      AN    DB94.DBX 133.7;
      =     L 6.0;
      A     L 6.0;
      L     DB94.DBW 134;
      SD    T 150;
      NOP   0;
      NOP   0;
      NOP   0;
      NOP   0;
      A     L 6.0;
      A     T 150;
      =     L 6.1;
      A     L 6.1;
      A(;
      O(;
      L     DB94.DBW 136;
      L     2;
      >=I;
      );
      O;
      AN    #PARAM5;
      AN    #PARAM6;
      );
      S     #PARAM23;
      A     L 6.1;
      A(;
      O     #PARAM23;
      O;
      A     #PARAM5;
      A     #PARAM6;
      );
      AN    DB94.DBX 133.7;
      =     L 6.2;
      A     L 6.2;
      JNB   M039;
      L     13;
      T     DB94.DBW 120;
M039: NOP   0;
      A     L 6.2;
      BLD   102;
      S     DB94.DBX 133.7;
      A     L 6.1;
      A     #PARAM5;
      AN    #PARAM6;
      AN    DB94.DBX 133.7;
      =     L 6.2;
      A     L 6.2;
      BLD   102;
      S     #PARAM14;
      A     L 6.2;
      BLD   102;
      R     #PARAM15;
      A     L 6.2;
      BLD   102;
      S     #PARAM20;
      A     L 6.2;
      JNB   M040;
      L     11;
      T     DB94.DBW 120;
M040: NOP   0;
      A     L 6.2;
      BLD   102;
      S     DB94.DBX 133.7;
      A     L 6.2;
      JNB   M041;
      L     DB94.DBW 136;
      L     1;
      +I;
      T     DB94.DBW 136;
M041: NOP   0;
      A     L 6.1;
      AN    #PARAM5;
      A     #PARAM6;
      AN    DB94.DBX 133.7;
      =     L 6.2;
      A     L 6.2;
      BLD   102;
      S     #PARAM15;
      A     L 6.2;
      BLD   102;
      R     #PARAM14;
      A     L 6.2;
      BLD   102;
      S     #PARAM20;
      A     L 6.2;
      JNB   M042;
      L     12;
      T     DB94.DBW 120;
M042: NOP   0;
      A     L 6.2;
      BLD   102;
      S     DB94.DBX 133.7;
      A     L 6.2;
      JNB   M043;
      L     DB94.DBW 136;
      L     1;
      +I;
      T     DB94.DBW 136;
M043: NOP   0;
NETWORK
TITLE =
      A(;
      L     DB94.DBW 120;
      L     11;
      ==I;
      );
      AN    DB94.DBX 133.7;
      A     #PARAM6;
      =     L 6.0;
      A     L 6.0;
      BLD   102;
      R     #PARAM14;
      A     L 6.0;
      BLD   102;
      R     #PARAM20;
      A     L 6.0;
      JNB   M044;
      L     10;
      T     DB94.DBW 120;
M044: NOP   0;
      A     L 6.0;
      BLD   102;
      S     DB94.DBX 133.7;
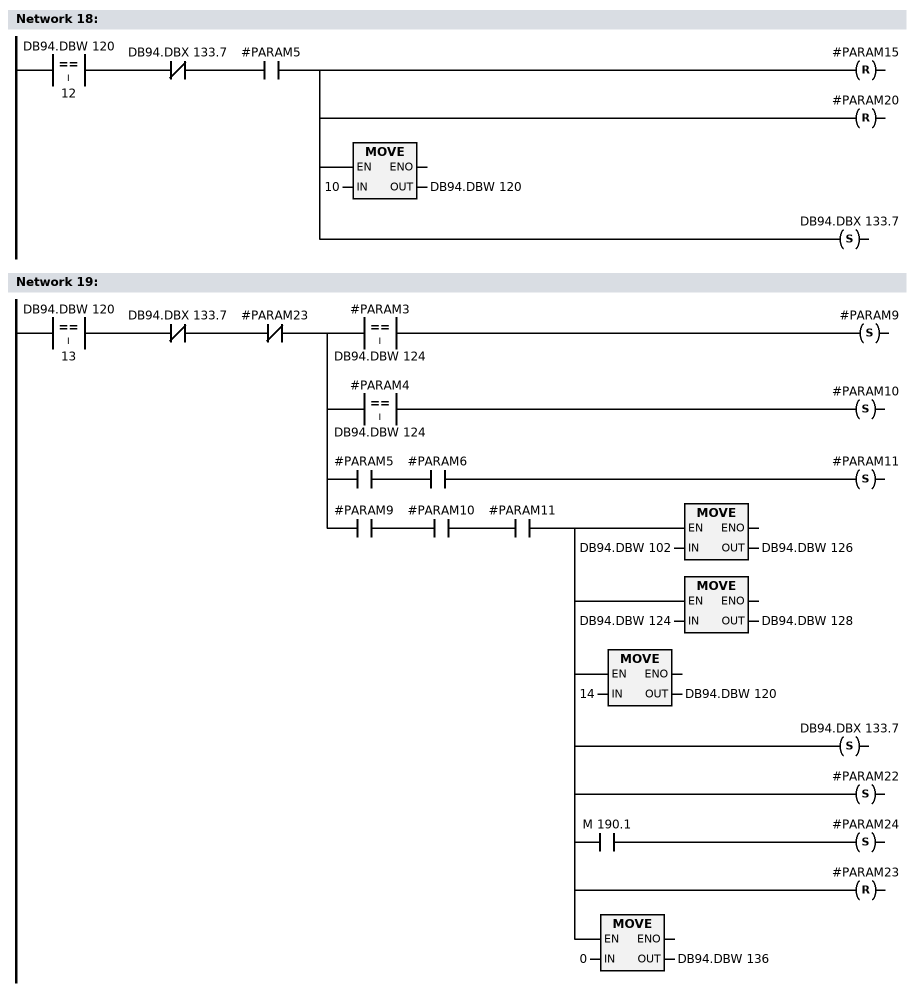
NETWORK
TITLE =
      A(;
      L     DB94.DBW 120;
      L     12;
      ==I;
      );
      AN    DB94.DBX 133.7;
      A     #PARAM5;
      =     L 6.0;
      A     L 6.0;
      BLD   102;
      R     #PARAM15;
      A     L 6.0;
      BLD   102;
      R     #PARAM20;
      A     L 6.0;
      JNB   M045;
      L     10;
      T     DB94.DBW 120;
M045: NOP   0;
      A     L 6.0;
      BLD   102;
      S     DB94.DBX 133.7;
NETWORK
TITLE =
      A(;
      L     DB94.DBW 120;
      L     13;
      ==I;
      );
      AN    DB94.DBX 133.7;
      AN    #PARAM23;
      =     L 6.0;
      A     L 6.0;
      A(;
      L     #PARAM3;
      L     DB94.DBW 124;
      ==I;
      );
      S     #PARAM9;
      A     L 6.0;
      A(;
      L     #PARAM4;
      L     DB94.DBW 124;
      ==I;
      );
      S     #PARAM10;
      A     L 6.0;
      A     #PARAM5;
      A     #PARAM6;
      S     #PARAM11;
      A     L 6.0;
      A     #PARAM9;
      A     #PARAM10;
      A     #PARAM11;
      =     L 6.1;
      A     L 6.1;
      JNB   M046;
      L     DB94.DBW 102;
      T     DB94.DBW 126;
M046: NOP   0;
      A     L 6.1;
      JNB   M047;
      L     DB94.DBW 124;
      T     DB94.DBW 128;
M047: NOP   0;
      A     L 6.1;
      JNB   M048;
      L     14;
      T     DB94.DBW 120;
M048: NOP   0;
      A     L 6.1;
      BLD   102;
      S     DB94.DBX 133.7;
      A     L 6.1;
      BLD   102;
      S     #PARAM22;
      A     L 6.1;
      A     M 190.1;
      S     #PARAM24;
      A     L 6.1;
      BLD   102;
      R     #PARAM23;
      A     L 6.1;
      JNB   M049;
      L     0;
      T     DB94.DBW 136;
M049: NOP   0;
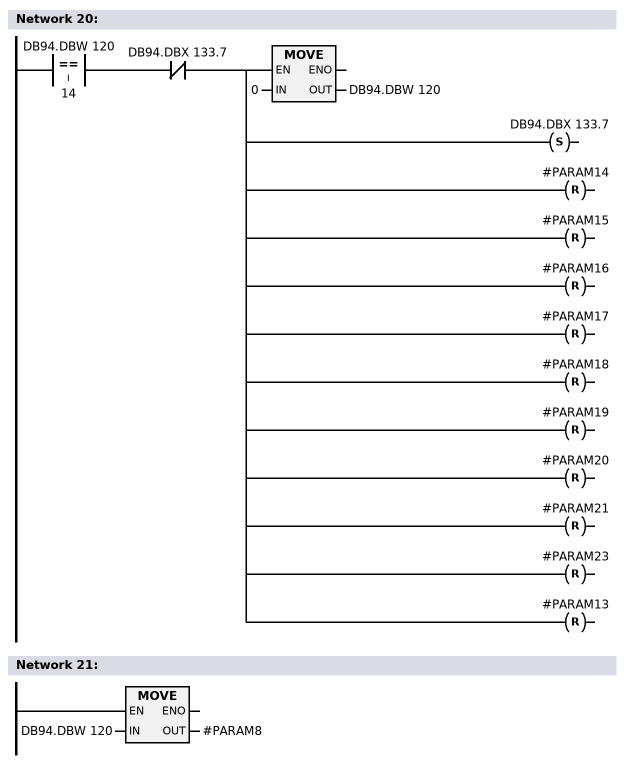
NETWORK
TITLE =
      A(;
      L     DB94.DBW 120;
      L     14;
      ==I;
      );
      AN    DB94.DBX 133.7;
      =     L 6.0;
      A     L 6.0;
      JNB   M050;
      L     0;
      T     DB94.DBW 120;
M050: NOP   0;
      A     L 6.0;
      BLD   102;
      S     DB94.DBX 133.7;
      A     L 6.0;
      BLD   102;
      R     #PARAM14;
      A     L 6.0;
      BLD   102;
      R     #PARAM15;
      A     L 6.0;
      BLD   102;
      R     #PARAM16;
      A     L 6.0;
      BLD   102;
      R     #PARAM17;
      A     L 6.0;
      BLD   102;
      R     #PARAM18;
      A     L 6.0;
      BLD   102;
      R     #PARAM19;
      A     L 6.0;
      BLD   102;
      R     #PARAM20;
      A     L 6.0;
      BLD   102;
      R     #PARAM21;
      A     L 6.0;
      BLD   102;
      R     #PARAM23;
      A     L 6.0;
      BLD   102;
      R     #PARAM13;
NETWORK
TITLE =
      L     DB94.DBW 120;
      T     #PARAM8;
      NOP   0;
END_FUNCTION

FUNCTION FC 95 : VOID
AUTHOR : SKD
FAMILY : AuTiPosi
NAME : CDSPL
VERSION : 0.1
BEGIN
// (block stored without names or comments; labels and parameter names are numbered)
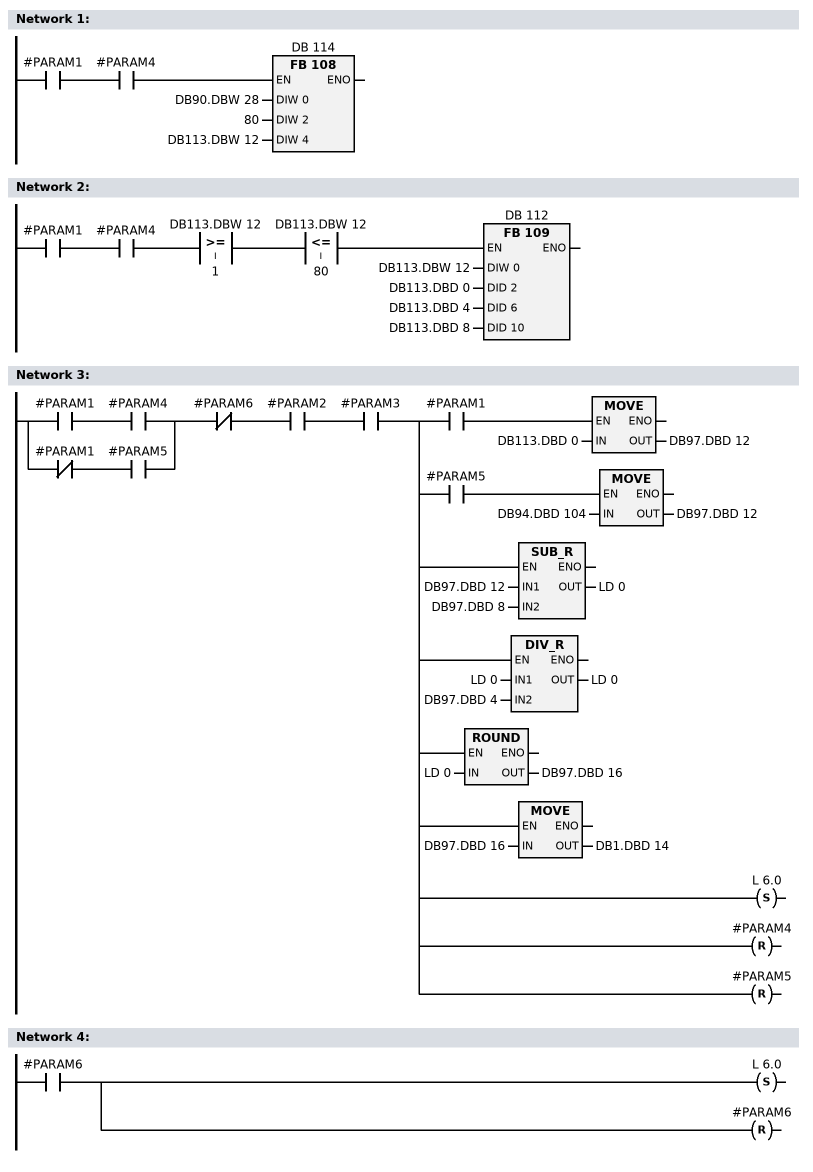
NETWORK
TITLE =
      A     #PARAM1;
      A     #PARAM4;
      JNB   M001;
      CALL  FB 108 , DB 114 (
           DIW 0                    := DB90.DBW 28,
           DIW 2                    := 80,
           DIW 4                    := DB113.DBW 12);
M001: NOP   0;
NETWORK
TITLE =
      A     #PARAM1;
      A     #PARAM4;
      A(;
      L     DB113.DBW 12;
      L     1;
      >=I;
      );
      A(;
      L     DB113.DBW 12;
      L     80;
      <=I;
      );
      JNB   M002;
      CALL  FB 109 , DB 112 (
           DIW 0                    := DB113.DBW 12,
           DID 2                    := DB113.DBD 0,
           DID 6                    := DB113.DBD 4,
           DID 10                   := DB113.DBD 8);
M002: NOP   0;
NETWORK
TITLE =
      A(;
      A     #PARAM1;
      A     #PARAM4;
      O;
      AN    #PARAM1;
      A     #PARAM5;
      );
      AN    #PARAM6;
      A     #PARAM2;
      A     #PARAM3;
      =     L 7.0;
      A     L 7.0;
      A     #PARAM1;
      JNB   M003;
      L     DB113.DBD 0;
      T     DB97.DBD 12;
M003: NOP   0;
      A     L 7.0;
      A     #PARAM5;
      JNB   M004;
      L     DB94.DBD 104;
      T     DB97.DBD 12;
M004: NOP   0;
      A     L 7.0;
      JNB   M005;
      L     DB97.DBD 12;
      L     DB97.DBD 8;
      -R;
      T     LD 0;
M005: NOP   0;
      A     L 7.0;
      JNB   M006;
      L     LD 0;
      L     DB97.DBD 4;
      /R;
      T     LD 0;
M006: NOP   0;
      A     L 7.0;
      JNB   M007;
      L     LD 0;
      RND;
      T     DB97.DBD 16;
M007: NOP   0;
      A     L 7.0;
      JNB   M008;
      L     DB97.DBD 16;
      T     DB1.DBD 14;
M008: NOP   0;
      A     L 7.0;
      BLD   102;
      S     L 6.0;
      A     L 7.0;
      BLD   102;
      R     #PARAM4;
      A     L 7.0;
      BLD   102;
      R     #PARAM5;
NETWORK
TITLE =
      A     #PARAM6;
      S     L 6.0;
      R     #PARAM6;
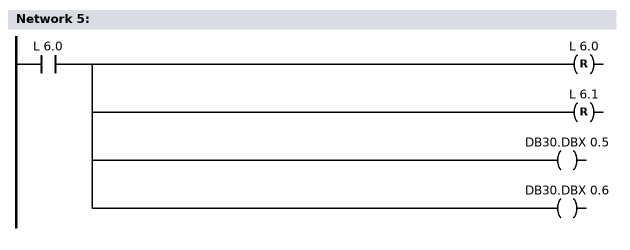
NETWORK
TITLE =
      A     L 6.0;
      R     L 6.0;
      R     L 6.1;
      =     DB30.DBX 0.5;
      =     DB30.DBX 0.6;
END_FUNCTION

FUNCTION FC 97 : VOID
AUTHOR : SKD
FAMILY : AuTiPosi
NAME : CDSPL
VERSION : 0.1
BEGIN
// (block stored without names or comments; labels and parameter names are numbered)
